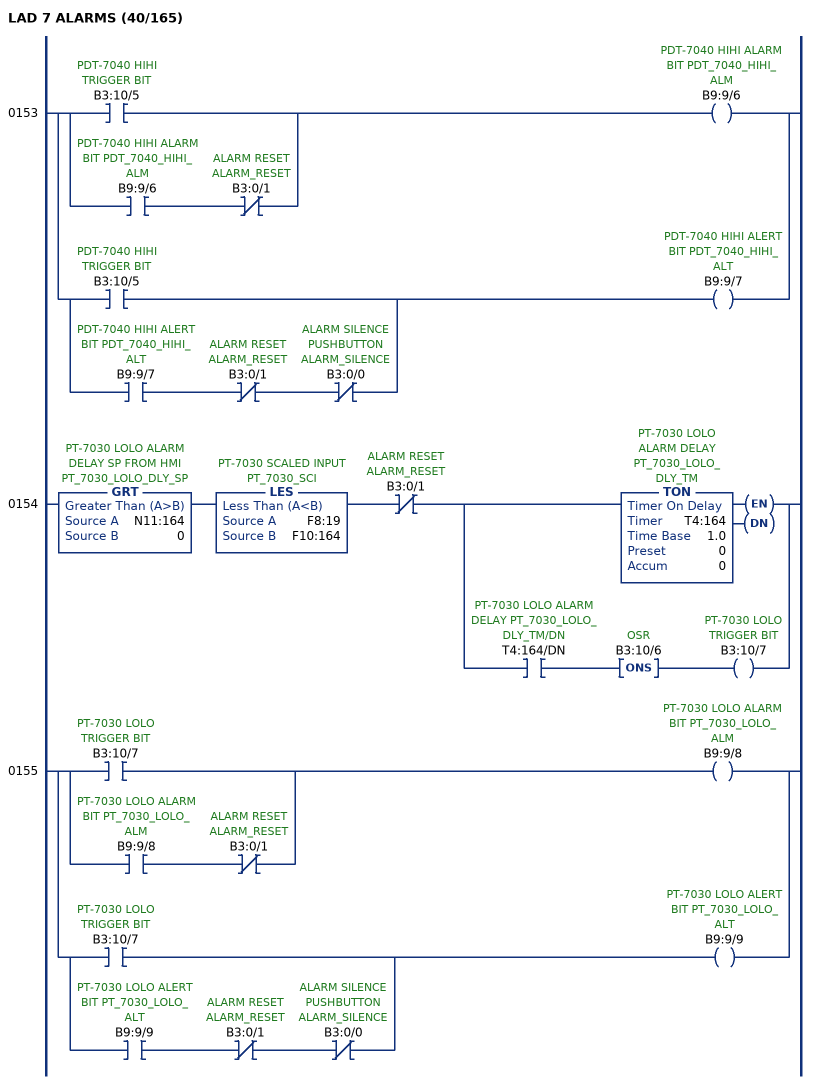
% Rung: 153 %
SOR BST BST XIC B3:10/5 NXB XIC B9:9/6 XIO B3:0/1 BND OTE B9:9/6 NXB BST XIC B3:10/5 NXB XIC B9:9/7 XIO B3:0/1 XIO B3:0/0 BND OTE B9:9/7 BND EOR
%   B3:10/5  "PDT-7040 HIHI TRIGGER BIT" %
%   B9:9/6  PDT_7040_HIHI_ALM  "PDT-7040 HIHI ALARM BIT" %
%   B3:0/1  ALARM_RESET  "ALARM RESET" %
%   B9:9/7  PDT_7040_HIHI_ALT  "PDT-7040 HIHI ALERT BIT" %
%   B3:0/0  ALARM_SILENCE  "ALARM SILENCE PUSHBUTTON" %
% Rung: 154 %
SOR GRT N11:164 0 LES F8:19 F10:164 XIO B3:0/1 BST TON T4:164 1.0 0 0 NXB XIC T4:164/DN OSR B3:10/6 OTE B3:10/7 BND EOR
%   N11:164  PT_7030_LOLO_DLY_SP  "PT-7030 LOLO ALARM DELAY SP FROM HMI" %
%   F8:19  PT_7030_SCI  "PT-7030 SCALED INPUT" %
%   F10:164  PT_7030_LOLO_SP  "PT-7030 LOLO ALARM SP" %
%   B3:0/1  ALARM_RESET  "ALARM RESET" %
%   T4:164  PT_7030_LOLO_DLY_TM  "PT-7030 LOLO ALARM DELAY" %
%   B3:10/6  "OSR" %
%   B3:10/7  "PT-7030 LOLO TRIGGER BIT" %
% Rung: 155 %
SOR BST BST XIC B3:10/7 NXB XIC B9:9/8 XIO B3:0/1 BND OTE B9:9/8 NXB BST XIC B3:10/7 NXB XIC B9:9/9 XIO B3:0/1 XIO B3:0/0 BND OTE B9:9/9 BND EOR
%   B3:10/7  "PT-7030 LOLO TRIGGER BIT" %
%   B9:9/8  PT_7030_LOLO_ALM  "PT-7030 LOLO ALARM BIT" %
%   B3:0/1  ALARM_RESET  "ALARM RESET" %
%   B9:9/9  PT_7030_LOLO_ALT  "PT-7030 LOLO ALERT BIT" %
%   B3:0/0  ALARM_SILENCE  "ALARM SILENCE PUSHBUTTON" %

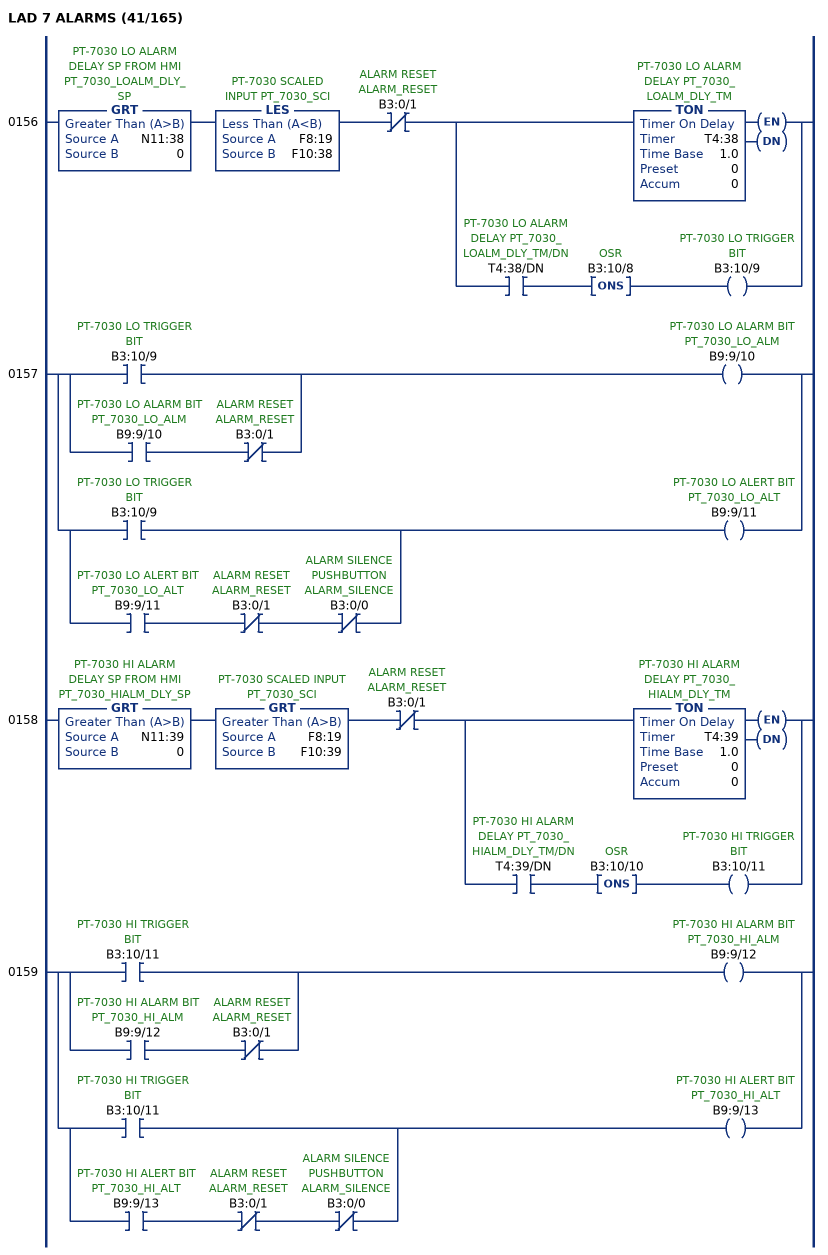
% Rung: 156 %
SOR GRT N11:38 0 LES F8:19 F10:38 XIO B3:0/1 BST TON T4:38 1.0 0 0 NXB XIC T4:38/DN OSR B3:10/8 OTE B3:10/9 BND EOR
%   N11:38  PT_7030_LOALM_DLY_SP  "PT-7030 LO ALARM DELAY SP FROM HMI" %
%   F8:19  PT_7030_SCI  "PT-7030 SCALED INPUT" %
%   F10:38  PT_7030_LOALM_SP  "PT-7030 LO ALARM SP" %
%   B3:0/1  ALARM_RESET  "ALARM RESET" %
%   T4:38  PT_7030_LOALM_DLY_TM  "PT-7030 LO ALARM DELAY" %
%   B3:10/8  "OSR" %
%   B3:10/9  "PT-7030 LO TRIGGER BIT" %
% Rung: 157 %
SOR BST BST XIC B3:10/9 NXB XIC B9:9/10 XIO B3:0/1 BND OTE B9:9/10 NXB BST XIC B3:10/9 NXB XIC B9:9/11 XIO B3:0/1 XIO B3:0/0 BND OTE B9:9/11 BND EOR
%   B3:10/9  "PT-7030 LO TRIGGER BIT" %
%   B9:9/10  PT_7030_LO_ALM  "PT-7030 LO ALARM BIT" %
%   B3:0/1  ALARM_RESET  "ALARM RESET" %
%   B9:9/11  PT_7030_LO_ALT  "PT-7030 LO ALERT BIT" %
%   B3:0/0  ALARM_SILENCE  "ALARM SILENCE PUSHBUTTON" %
% Rung: 158 %
SOR GRT N11:39 0 GRT F8:19 F10:39 XIO B3:0/1 BST TON T4:39 1.0 0 0 NXB XIC T4:39/DN OSR B3:10/10 OTE B3:10/11 BND EOR
%   N11:39  PT_7030_HIALM_DLY_SP  "PT-7030 HI ALARM DELAY SP FROM HMI" %
%   F8:19  PT_7030_SCI  "PT-7030 SCALED INPUT" %
%   F10:39  PT_7030_HIALM_SP  "PT-7030 HI ALARM SP" %
%   B3:0/1  ALARM_RESET  "ALARM RESET" %
%   T4:39  PT_7030_HIALM_DLY_TM  "PT-7030 HI ALARM DELAY" %
%   B3:10/10  "OSR" %
%   B3:10/11  "PT-7030 HI TRIGGER BIT" %
% Rung: 159 %
SOR BST BST XIC B3:10/11 NXB XIC B9:9/12 XIO B3:0/1 BND OTE B9:9/12 NXB BST XIC B3:10/11 NXB XIC B9:9/13 XIO B3:0/1 XIO B3:0/0 BND OTE B9:9/13 BND EOR
%   B3:10/11  "PT-7030 HI TRIGGER BIT" %
%   B9:9/12  PT_7030_HI_ALM  "PT-7030 HI ALARM BIT" %
%   B3:0/1  ALARM_RESET  "ALARM RESET" %
%   B9:9/13  PT_7030_HI_ALT  "PT-7030 HI ALERT BIT" %
%   B3:0/0  ALARM_SILENCE  "ALARM SILENCE PUSHBUTTON" %

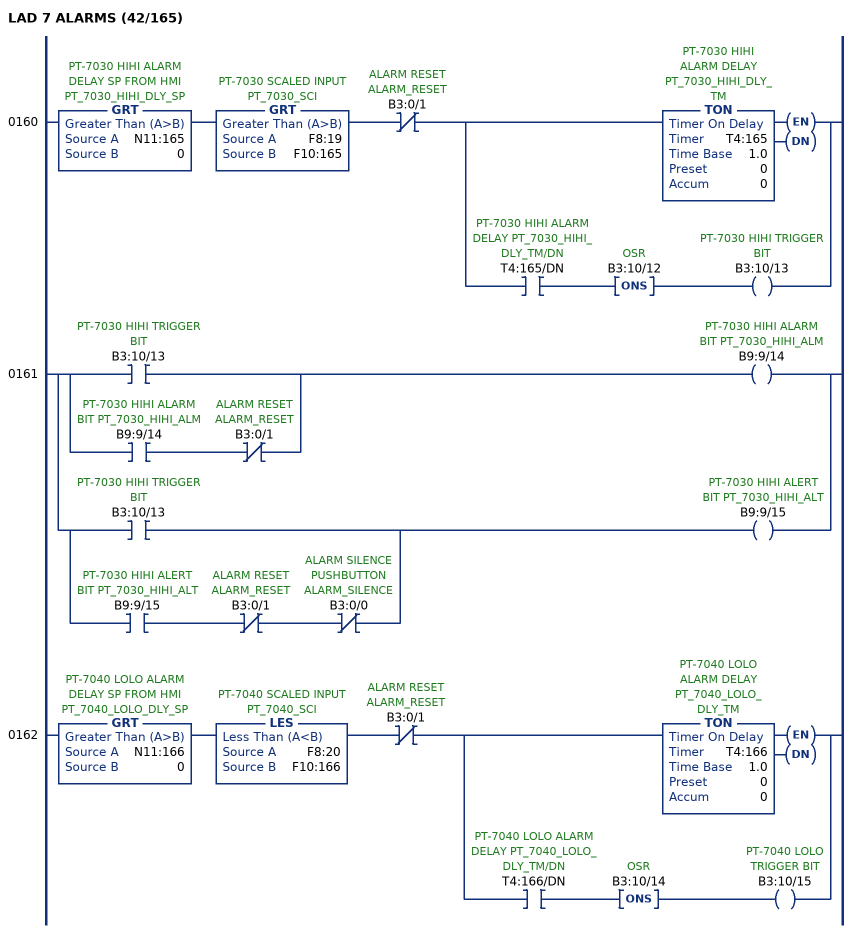
% Rung: 160 %
SOR GRT N11:165 0 GRT F8:19 F10:165 XIO B3:0/1 BST TON T4:165 1.0 0 0 NXB XIC T4:165/DN OSR B3:10/12 OTE B3:10/13 BND EOR
%   N11:165  PT_7030_HIHI_DLY_SP  "PT-7030 HIHI ALARM DELAY SP FROM HMI" %
%   F8:19  PT_7030_SCI  "PT-7030 SCALED INPUT" %
%   F10:165  PT_7030_HIHI_SP  "PT-7030 HIHI ALARM SP" %
%   B3:0/1  ALARM_RESET  "ALARM RESET" %
%   T4:165  PT_7030_HIHI_DLY_TM  "PT-7030 HIHI ALARM DELAY" %
%   B3:10/12  "OSR" %
%   B3:10/13  "PT-7030 HIHI TRIGGER BIT" %
% Rung: 161 %
SOR BST BST XIC B3:10/13 NXB XIC B9:9/14 XIO B3:0/1 BND OTE B9:9/14 NXB BST XIC B3:10/13 NXB XIC B9:9/15 XIO B3:0/1 XIO B3:0/0 BND OTE B9:9/15 BND EOR
%   B3:10/13  "PT-7030 HIHI TRIGGER BIT" %
%   B9:9/14  PT_7030_HIHI_ALM  "PT-7030 HIHI ALARM BIT" %
%   B3:0/1  ALARM_RESET  "ALARM RESET" %
%   B9:9/15  PT_7030_HIHI_ALT  "PT-7030 HIHI ALERT BIT" %
%   B3:0/0  ALARM_SILENCE  "ALARM SILENCE PUSHBUTTON" %
% Rung: 162 %
SOR GRT N11:166 0 LES F8:20 F10:166 XIO B3:0/1 BST TON T4:166 1.0 0 0 NXB XIC T4:166/DN OSR B3:10/14 OTE B3:10/15 BND EOR
%   N11:166  PT_7040_LOLO_DLY_SP  "PT-7040 LOLO ALARM DELAY SP FROM HMI" %
%   F8:20  PT_7040_SCI  "PT-7040 SCALED INPUT" %
%   F10:166  PT_7040_LOLO_SP  "PT-7040 LOLO ALARM SP" %
%   B3:0/1  ALARM_RESET  "ALARM RESET" %
%   T4:166  PT_7040_LOLO_DLY_TM  "PT-7040 LOLO ALARM DELAY" %
%   B3:10/14  "OSR" %
%   B3:10/15  "PT-7040 LOLO TRIGGER BIT" %

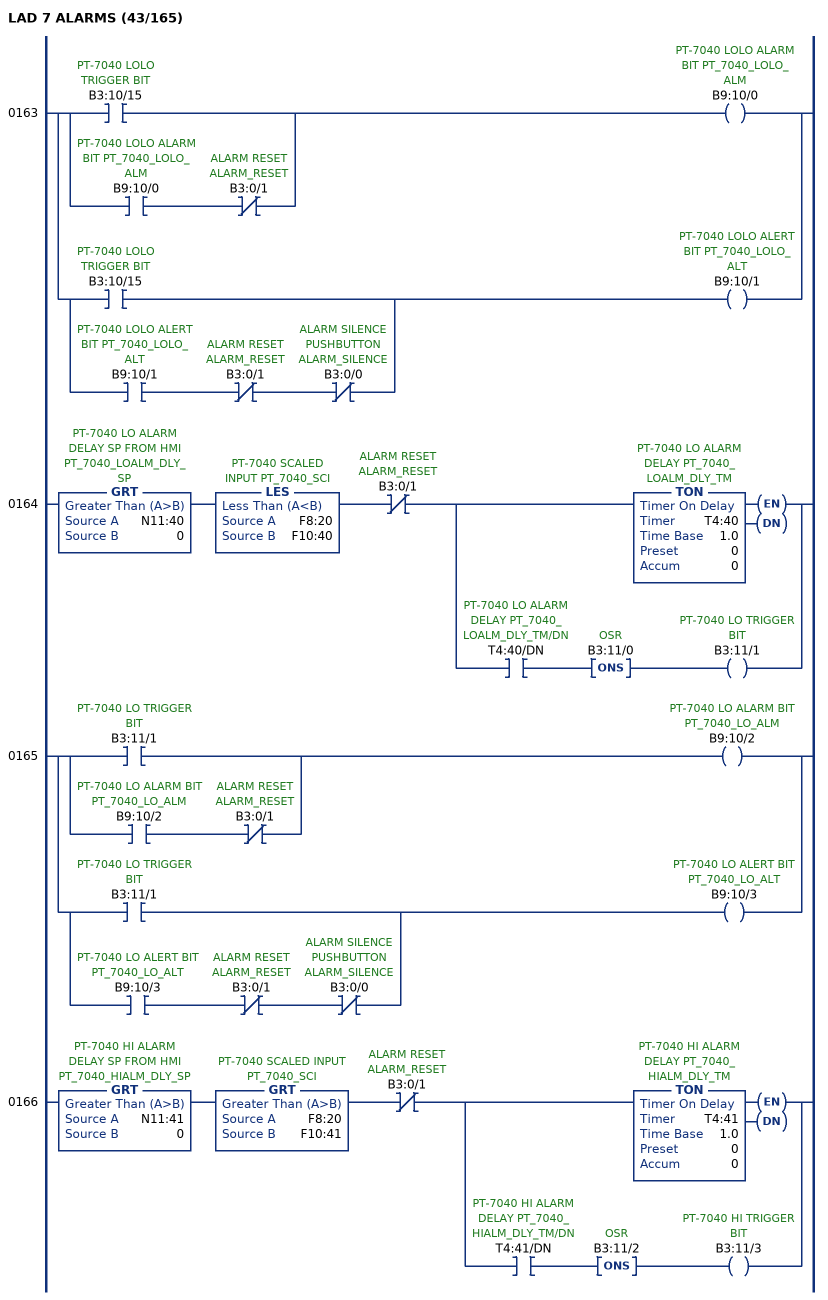
% Rung: 163 %
SOR BST BST XIC B3:10/15 NXB XIC B9:10/0 XIO B3:0/1 BND OTE B9:10/0 NXB BST XIC B3:10/15 NXB XIC B9:10/1 XIO B3:0/1 XIO B3:0/0 BND OTE B9:10/1 BND EOR
%   B3:10/15  "PT-7040 LOLO TRIGGER BIT" %
%   B9:10/0  PT_7040_LOLO_ALM  "PT-7040 LOLO ALARM BIT" %
%   B3:0/1  ALARM_RESET  "ALARM RESET" %
%   B9:10/1  PT_7040_LOLO_ALT  "PT-7040 LOLO ALERT BIT" %
%   B3:0/0  ALARM_SILENCE  "ALARM SILENCE PUSHBUTTON" %
% Rung: 164 %
SOR GRT N11:40 0 LES F8:20 F10:40 XIO B3:0/1 BST TON T4:40 1.0 0 0 NXB XIC T4:40/DN OSR B3:11/0 OTE B3:11/1 BND EOR
%   N11:40  PT_7040_LOALM_DLY_SP  "PT-7040 LO ALARM DELAY SP FROM HMI" %
%   F8:20  PT_7040_SCI  "PT-7040 SCALED INPUT" %
%   F10:40  PT_7040_LOALM_SP  "PT-7040 LO ALARM SP" %
%   B3:0/1  ALARM_RESET  "ALARM RESET" %
%   T4:40  PT_7040_LOALM_DLY_TM  "PT-7040 LO ALARM DELAY" %
%   B3:11/0  "OSR" %
%   B3:11/1  "PT-7040 LO TRIGGER BIT" %
% Rung: 165 %
SOR BST BST XIC B3:11/1 NXB XIC B9:10/2 XIO B3:0/1 BND OTE B9:10/2 NXB BST XIC B3:11/1 NXB XIC B9:10/3 XIO B3:0/1 XIO B3:0/0 BND OTE B9:10/3 BND EOR
%   B3:11/1  "PT-7040 LO TRIGGER BIT" %
%   B9:10/2  PT_7040_LO_ALM  "PT-7040 LO ALARM BIT" %
%   B3:0/1  ALARM_RESET  "ALARM RESET" %
%   B9:10/3  PT_7040_LO_ALT  "PT-7040 LO ALERT BIT" %
%   B3:0/0  ALARM_SILENCE  "ALARM SILENCE PUSHBUTTON" %
% Rung: 166 %
SOR GRT N11:41 0 GRT F8:20 F10:41 XIO B3:0/1 BST TON T4:41 1.0 0 0 NXB XIC T4:41/DN OSR B3:11/2 OTE B3:11/3 BND EOR
%   N11:41  PT_7040_HIALM_DLY_SP  "PT-7040 HI ALARM DELAY SP FROM HMI" %
%   F8:20  PT_7040_SCI  "PT-7040 SCALED INPUT" %
%   F10:41  PT_7040_HIALM_SP  "PT-7040 HI ALARM SP" %
%   B3:0/1  ALARM_RESET  "ALARM RESET" %
%   T4:41  PT_7040_HIALM_DLY_TM  "PT-7040 HI ALARM DELAY" %
%   B3:11/2  "OSR" %
%   B3:11/3  "PT-7040 HI TRIGGER BIT" %

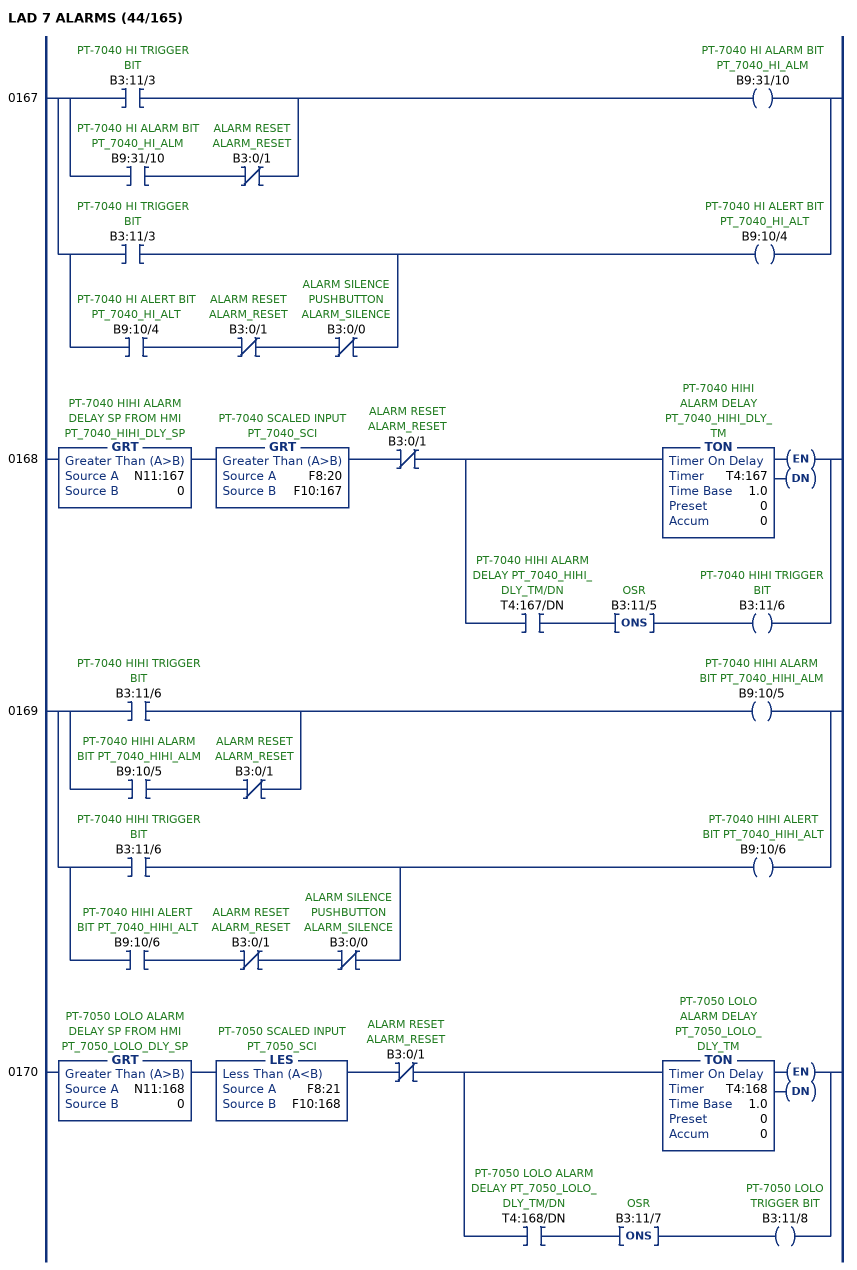
% Rung: 167 %
SOR BST BST XIC B3:11/3 NXB XIC B9:31/10 XIO B3:0/1 BND OTE B9:31/10 NXB BST XIC B3:11/3 NXB XIC B9:10/4 XIO B3:0/1 XIO B3:0/0 BND OTE B9:10/4 BND EOR
%   B3:11/3  "PT-7040 HI TRIGGER BIT" %
%   B9:31/10  PT_7040_HI_ALM  "PT-7040 HI ALARM BIT" %
%   B3:0/1  ALARM_RESET  "ALARM RESET" %
%   B9:10/4  PT_7040_HI_ALT  "PT-7040 HI ALERT BIT" %
%   B3:0/0  ALARM_SILENCE  "ALARM SILENCE PUSHBUTTON" %
% Rung: 168 %
SOR GRT N11:167 0 GRT F8:20 F10:167 XIO B3:0/1 BST TON T4:167 1.0 0 0 NXB XIC T4:167/DN OSR B3:11/5 OTE B3:11/6 BND EOR
%   N11:167  PT_7040_HIHI_DLY_SP  "PT-7040 HIHI ALARM DELAY SP FROM HMI" %
%   F8:20  PT_7040_SCI  "PT-7040 SCALED INPUT" %
%   F10:167  PT_7040_HIHI_SP  "PT-7040 HIHI ALARM SP" %
%   B3:0/1  ALARM_RESET  "ALARM RESET" %
%   T4:167  PT_7040_HIHI_DLY_TM  "PT-7040 HIHI ALARM DELAY" %
%   B3:11/5  "OSR" %
%   B3:11/6  "PT-7040 HIHI TRIGGER BIT" %
% Rung: 169 %
SOR BST BST XIC B3:11/6 NXB XIC B9:10/5 XIO B3:0/1 BND OTE B9:10/5 NXB BST XIC B3:11/6 NXB XIC B9:10/6 XIO B3:0/1 XIO B3:0/0 BND OTE B9:10/6 BND EOR
%   B3:11/6  "PT-7040 HIHI TRIGGER BIT" %
%   B9:10/5  PT_7040_HIHI_ALM  "PT-7040 HIHI ALARM BIT" %
%   B3:0/1  ALARM_RESET  "ALARM RESET" %
%   B9:10/6  PT_7040_HIHI_ALT  "PT-7040 HIHI ALERT BIT" %
%   B3:0/0  ALARM_SILENCE  "ALARM SILENCE PUSHBUTTON" %
% Rung: 170 %
SOR GRT N11:168 0 LES F8:21 F10:168 XIO B3:0/1 BST TON T4:168 1.0 0 0 NXB XIC T4:168/DN OSR B3:11/7 OTE B3:11/8 BND EOR
%   N11:168  PT_7050_LOLO_DLY_SP  "PT-7050 LOLO ALARM DELAY SP FROM HMI" %
%   F8:21  PT_7050_SCI  "PT-7050 SCALED INPUT" %
%   F10:168  PT_7050_LOLO_SP  "PT-7050 LOLO ALARM SP" %
%   B3:0/1  ALARM_RESET  "ALARM RESET" %
%   T4:168  PT_7050_LOLO_DLY_TM  "PT-7050 LOLO ALARM DELAY" %
%   B3:11/7  "OSR" %
%   B3:11/8  "PT-7050 LOLO TRIGGER BIT" %

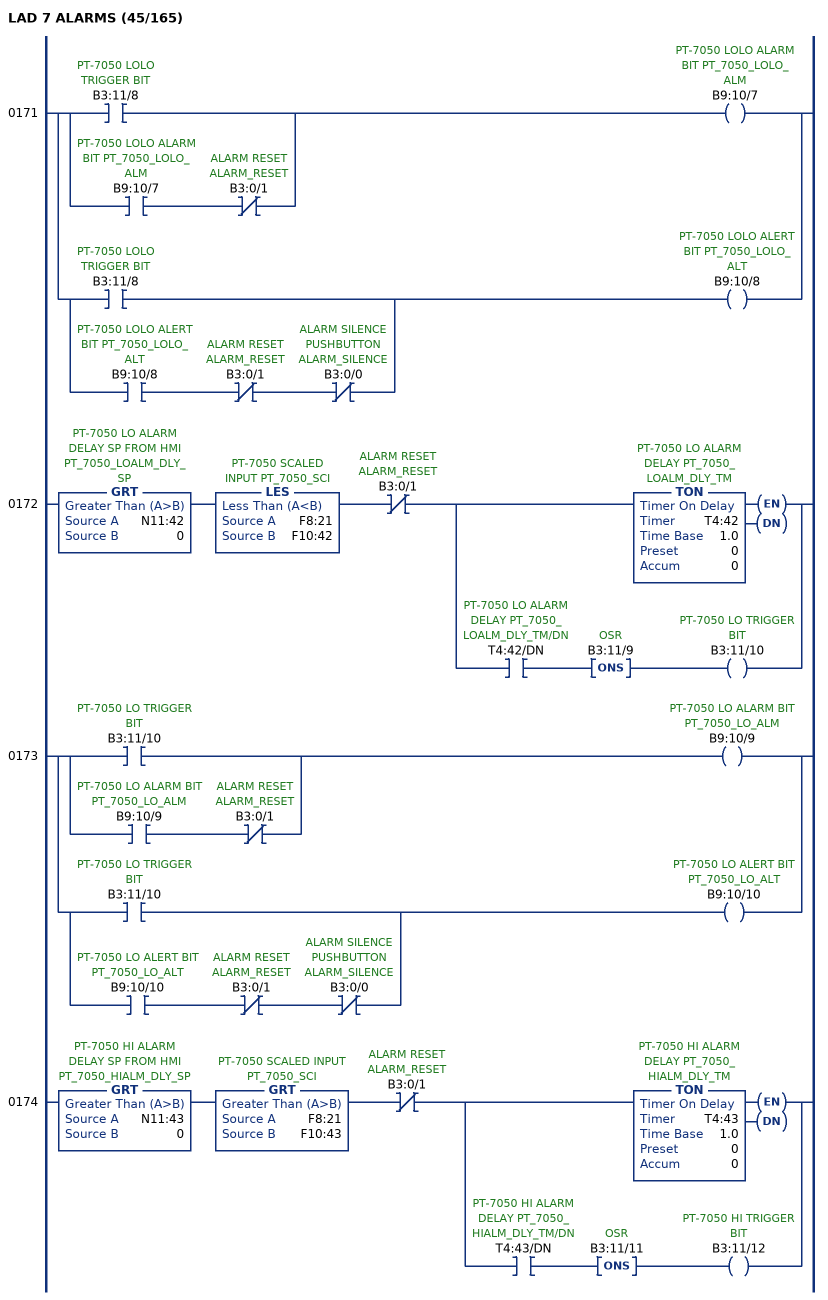
% Rung: 171 %
SOR BST BST XIC B3:11/8 NXB XIC B9:10/7 XIO B3:0/1 BND OTE B9:10/7 NXB BST XIC B3:11/8 NXB XIC B9:10/8 XIO B3:0/1 XIO B3:0/0 BND OTE B9:10/8 BND EOR
%   B3:11/8  "PT-7050 LOLO TRIGGER BIT" %
%   B9:10/7  PT_7050_LOLO_ALM  "PT-7050 LOLO ALARM BIT" %
%   B3:0/1  ALARM_RESET  "ALARM RESET" %
%   B9:10/8  PT_7050_LOLO_ALT  "PT-7050 LOLO ALERT BIT" %
%   B3:0/0  ALARM_SILENCE  "ALARM SILENCE PUSHBUTTON" %
% Rung: 172 %
SOR GRT N11:42 0 LES F8:21 F10:42 XIO B3:0/1 BST TON T4:42 1.0 0 0 NXB XIC T4:42/DN OSR B3:11/9 OTE B3:11/10 BND EOR
%   N11:42  PT_7050_LOALM_DLY_SP  "PT-7050 LO ALARM DELAY SP FROM HMI" %
%   F8:21  PT_7050_SCI  "PT-7050 SCALED INPUT" %
%   F10:42  PT_7050_LOALM_SP  "PT-7050 LO ALARM SP" %
%   B3:0/1  ALARM_RESET  "ALARM RESET" %
%   T4:42  PT_7050_LOALM_DLY_TM  "PT-7050 LO ALARM DELAY" %
%   B3:11/9  "OSR" %
%   B3:11/10  "PT-7050 LO TRIGGER BIT" %
% Rung: 173 %
SOR BST BST XIC B3:11/10 NXB XIC B9:10/9 XIO B3:0/1 BND OTE B9:10/9 NXB BST XIC B3:11/10 NXB XIC B9:10/10 XIO B3:0/1 XIO B3:0/0 BND OTE B9:10/10 BND EOR
%   B3:11/10  "PT-7050 LO TRIGGER BIT" %
%   B9:10/9  PT_7050_LO_ALM  "PT-7050 LO ALARM BIT" %
%   B3:0/1  ALARM_RESET  "ALARM RESET" %
%   B9:10/10  PT_7050_LO_ALT  "PT-7050 LO ALERT BIT" %
%   B3:0/0  ALARM_SILENCE  "ALARM SILENCE PUSHBUTTON" %
% Rung: 174 %
SOR GRT N11:43 0 GRT F8:21 F10:43 XIO B3:0/1 BST TON T4:43 1.0 0 0 NXB XIC T4:43/DN OSR B3:11/11 OTE B3:11/12 BND EOR
%   N11:43  PT_7050_HIALM_DLY_SP  "PT-7050 HI ALARM DELAY SP FROM HMI" %
%   F8:21  PT_7050_SCI  "PT-7050 SCALED INPUT" %
%   F10:43  PT_7050_HIALM_SP  "PT-7050 HI ALARM SP" %
%   B3:0/1  ALARM_RESET  "ALARM RESET" %
%   T4:43  PT_7050_HIALM_DLY_TM  "PT-7050 HI ALARM DELAY" %
%   B3:11/11  "OSR" %
%   B3:11/12  "PT-7050 HI TRIGGER BIT" %

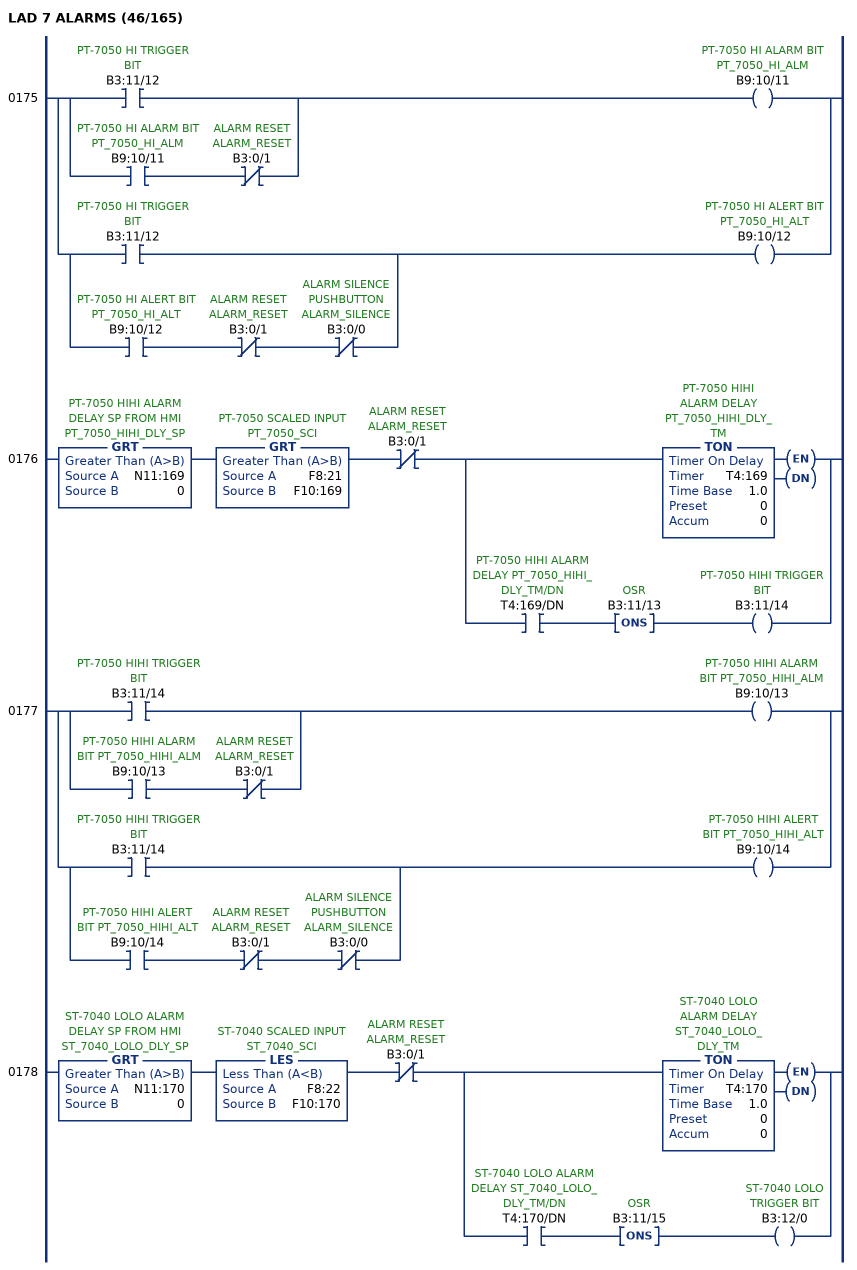
% Rung: 175 %
SOR BST BST XIC B3:11/12 NXB XIC B9:10/11 XIO B3:0/1 BND OTE B9:10/11 NXB BST XIC B3:11/12 NXB XIC B9:10/12 XIO B3:0/1 XIO B3:0/0 BND OTE B9:10/12 BND EOR
%   B3:11/12  "PT-7050 HI TRIGGER BIT" %
%   B9:10/11  PT_7050_HI_ALM  "PT-7050 HI ALARM BIT" %
%   B3:0/1  ALARM_RESET  "ALARM RESET" %
%   B9:10/12  PT_7050_HI_ALT  "PT-7050 HI ALERT BIT" %
%   B3:0/0  ALARM_SILENCE  "ALARM SILENCE PUSHBUTTON" %
% Rung: 176 %
SOR GRT N11:169 0 GRT F8:21 F10:169 XIO B3:0/1 BST TON T4:169 1.0 0 0 NXB XIC T4:169/DN OSR B3:11/13 OTE B3:11/14 BND EOR
%   N11:169  PT_7050_HIHI_DLY_SP  "PT-7050 HIHI ALARM DELAY SP FROM HMI" %
%   F8:21  PT_7050_SCI  "PT-7050 SCALED INPUT" %
%   F10:169  PT_7050_HIHI_SP  "PT-7050 HIHI ALARM SP" %
%   B3:0/1  ALARM_RESET  "ALARM RESET" %
%   T4:169  PT_7050_HIHI_DLY_TM  "PT-7050 HIHI ALARM DELAY" %
%   B3:11/13  "OSR" %
%   B3:11/14  "PT-7050 HIHI TRIGGER BIT" %
% Rung: 177 %
SOR BST BST XIC B3:11/14 NXB XIC B9:10/13 XIO B3:0/1 BND OTE B9:10/13 NXB BST XIC B3:11/14 NXB XIC B9:10/14 XIO B3:0/1 XIO B3:0/0 BND OTE B9:10/14 BND EOR
%   B3:11/14  "PT-7050 HIHI TRIGGER BIT" %
%   B9:10/13  PT_7050_HIHI_ALM  "PT-7050 HIHI ALARM BIT" %
%   B3:0/1  ALARM_RESET  "ALARM RESET" %
%   B9:10/14  PT_7050_HIHI_ALT  "PT-7050 HIHI ALERT BIT" %
%   B3:0/0  ALARM_SILENCE  "ALARM SILENCE PUSHBUTTON" %
% Rung: 178 %
SOR GRT N11:170 0 LES F8:22 F10:170 XIO B3:0/1 BST TON T4:170 1.0 0 0 NXB XIC T4:170/DN OSR B3:11/15 OTE B3:12/0 BND EOR
%   N11:170  ST_7040_LOLO_DLY_SP  "ST-7040 LOLO ALARM DELAY SP FROM HMI" %
%   F8:22  ST_7040_SCI  "ST-7040 SCALED INPUT" %
%   F10:170  ST_7040_LOLO_SP  "ST-7040 LOLO ALARM SP" %
%   B3:0/1  ALARM_RESET  "ALARM RESET" %
%   T4:170  ST_7040_LOLO_DLY_TM  "ST-7040 LOLO ALARM DELAY" %
%   B3:11/15  "OSR" %
%   B3:12/0  "ST-7040 LOLO TRIGGER BIT" %

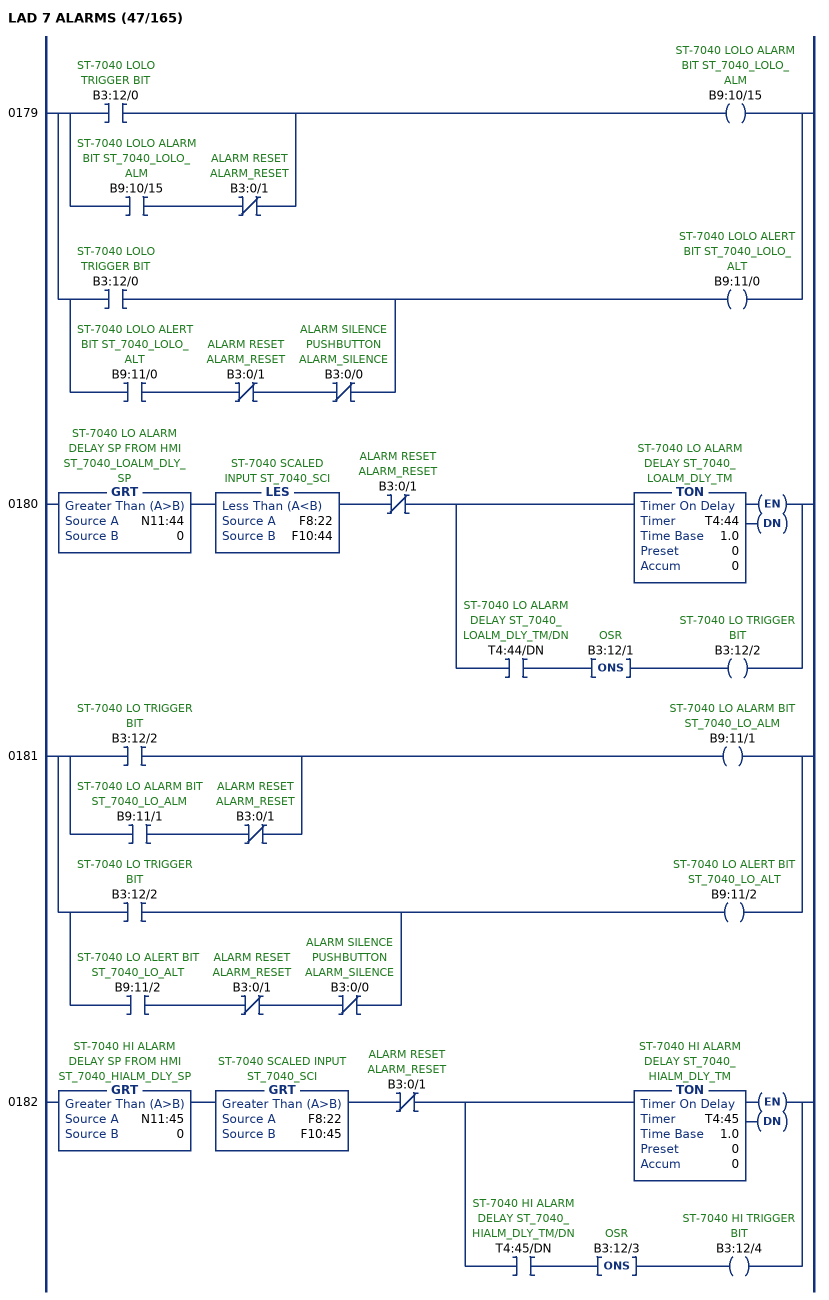
% Rung: 179 %
SOR BST BST XIC B3:12/0 NXB XIC B9:10/15 XIO B3:0/1 BND OTE B9:10/15 NXB BST XIC B3:12/0 NXB XIC B9:11/0 XIO B3:0/1 XIO B3:0/0 BND OTE B9:11/0 BND EOR
%   B3:12/0  "ST-7040 LOLO TRIGGER BIT" %
%   B9:10/15  ST_7040_LOLO_ALM  "ST-7040 LOLO ALARM BIT" %
%   B3:0/1  ALARM_RESET  "ALARM RESET" %
%   B9:11/0  ST_7040_LOLO_ALT  "ST-7040 LOLO ALERT BIT" %
%   B3:0/0  ALARM_SILENCE  "ALARM SILENCE PUSHBUTTON" %
% Rung: 180 %
SOR GRT N11:44 0 LES F8:22 F10:44 XIO B3:0/1 BST TON T4:44 1.0 0 0 NXB XIC T4:44/DN OSR B3:12/1 OTE B3:12/2 BND EOR
%   N11:44  ST_7040_LOALM_DLY_SP  "ST-7040 LO ALARM DELAY SP FROM HMI" %
%   F8:22  ST_7040_SCI  "ST-7040 SCALED INPUT" %
%   F10:44  ST_7040_LOALM_SP  "ST-7040 LO ALARM SP" %
%   B3:0/1  ALARM_RESET  "ALARM RESET" %
%   T4:44  ST_7040_LOALM_DLY_TM  "ST-7040 LO ALARM DELAY" %
%   B3:12/1  "OSR" %
%   B3:12/2  "ST-7040 LO TRIGGER BIT" %
% Rung: 181 %
SOR BST BST XIC B3:12/2 NXB XIC B9:11/1 XIO B3:0/1 BND OTE B9:11/1 NXB BST XIC B3:12/2 NXB XIC B9:11/2 XIO B3:0/1 XIO B3:0/0 BND OTE B9:11/2 BND EOR
%   B3:12/2  "ST-7040 LO TRIGGER BIT" %
%   B9:11/1  ST_7040_LO_ALM  "ST-7040 LO ALARM BIT" %
%   B3:0/1  ALARM_RESET  "ALARM RESET" %
%   B9:11/2  ST_7040_LO_ALT  "ST-7040 LO ALERT BIT" %
%   B3:0/0  ALARM_SILENCE  "ALARM SILENCE PUSHBUTTON" %
% Rung: 182 %
SOR GRT N11:45 0 GRT F8:22 F10:45 XIO B3:0/1 BST TON T4:45 1.0 0 0 NXB XIC T4:45/DN OSR B3:12/3 OTE B3:12/4 BND EOR
%   N11:45  ST_7040_HIALM_DLY_SP  "ST-7040 HI ALARM DELAY SP FROM HMI" %
%   F8:22  ST_7040_SCI  "ST-7040 SCALED INPUT" %
%   F10:45  ST_7040_HIALM_SP  "ST-7040 HI ALARM SP" %
%   B3:0/1  ALARM_RESET  "ALARM RESET" %
%   T4:45  ST_7040_HIALM_DLY_TM  "ST-7040 HI ALARM DELAY" %
%   B3:12/3  "OSR" %
%   B3:12/4  "ST-7040 HI TRIGGER BIT" %

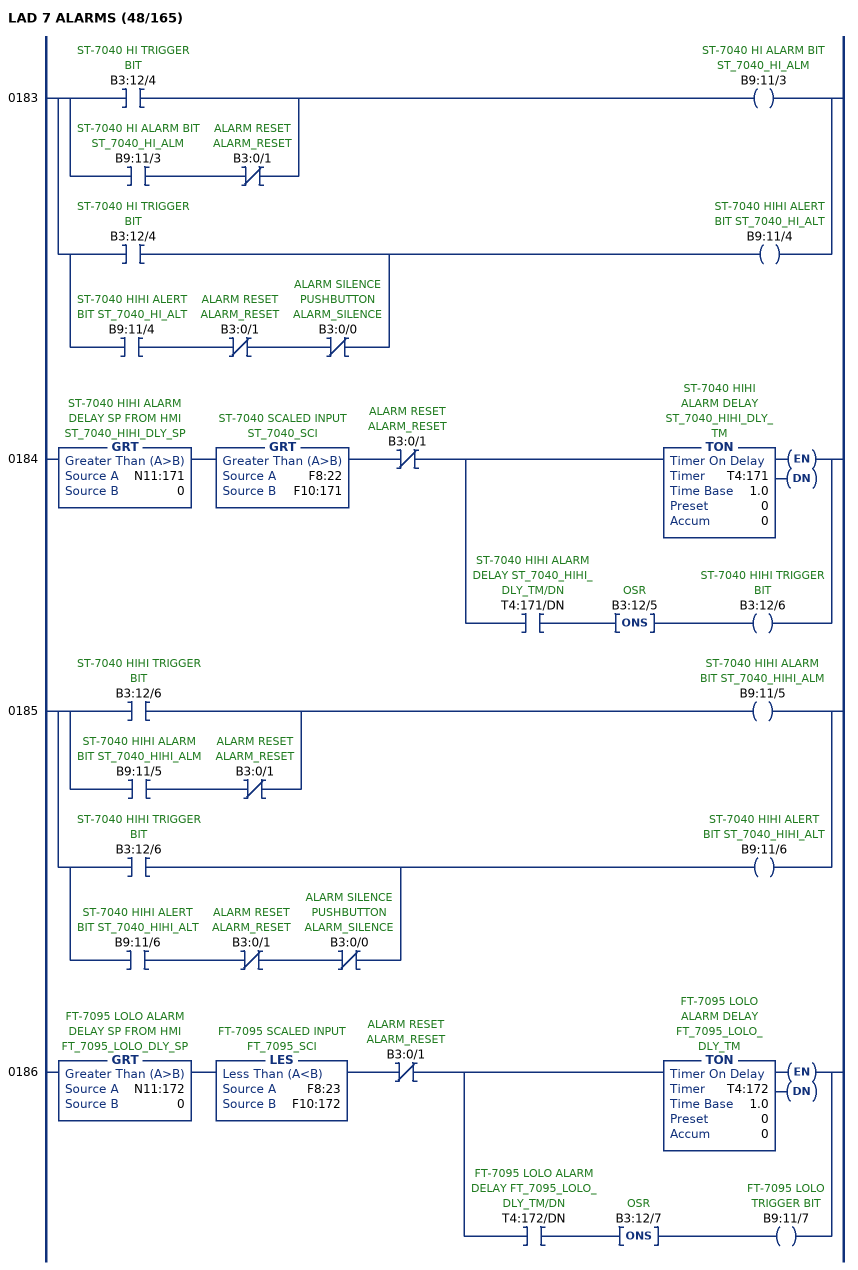
% Rung: 183 %
SOR BST BST XIC B3:12/4 NXB XIC B9:11/3 XIO B3:0/1 BND OTE B9:11/3 NXB BST XIC B3:12/4 NXB XIC B9:11/4 XIO B3:0/1 XIO B3:0/0 BND OTE B9:11/4 BND EOR
%   B3:12/4  "ST-7040 HI TRIGGER BIT" %
%   B9:11/3  ST_7040_HI_ALM  "ST-7040 HI ALARM BIT" %
%   B3:0/1  ALARM_RESET  "ALARM RESET" %
%   B9:11/4  ST_7040_HI_ALT  "ST-7040 HIHI ALERT BIT" %
%   B3:0/0  ALARM_SILENCE  "ALARM SILENCE PUSHBUTTON" %
% Rung: 184 %
SOR GRT N11:171 0 GRT F8:22 F10:171 XIO B3:0/1 BST TON T4:171 1.0 0 0 NXB XIC T4:171/DN OSR B3:12/5 OTE B3:12/6 BND EOR
%   N11:171  ST_7040_HIHI_DLY_SP  "ST-7040 HIHI ALARM DELAY SP FROM HMI" %
%   F8:22  ST_7040_SCI  "ST-7040 SCALED INPUT" %
%   F10:171  ST_7040_HIHI_SP  "ST-7040 HIHI ALARM SP" %
%   B3:0/1  ALARM_RESET  "ALARM RESET" %
%   T4:171  ST_7040_HIHI_DLY_TM  "ST-7040 HIHI ALARM DELAY" %
%   B3:12/5  "OSR" %
%   B3:12/6  "ST-7040 HIHI TRIGGER BIT" %
% Rung: 185 %
SOR BST BST XIC B3:12/6 NXB XIC B9:11/5 XIO B3:0/1 BND OTE B9:11/5 NXB BST XIC B3:12/6 NXB XIC B9:11/6 XIO B3:0/1 XIO B3:0/0 BND OTE B9:11/6 BND EOR
%   B3:12/6  "ST-7040 HIHI TRIGGER BIT" %
%   B9:11/5  ST_7040_HIHI_ALM  "ST-7040 HIHI ALARM BIT" %
%   B3:0/1  ALARM_RESET  "ALARM RESET" %
%   B9:11/6  ST_7040_HIHI_ALT  "ST-7040 HIHI ALERT BIT" %
%   B3:0/0  ALARM_SILENCE  "ALARM SILENCE PUSHBUTTON" %
% Rung: 186 %
SOR GRT N11:172 0 LES F8:23 F10:172 XIO B3:0/1 BST TON T4:172 1.0 0 0 NXB XIC T4:172/DN OSR B3:12/7 OTE B9:11/7 BND EOR
%   N11:172  FT_7095_LOLO_DLY_SP  "FT-7095 LOLO ALARM DELAY SP FROM HMI" %
%   F8:23  FT_7095_SCI  "FT-7095 SCALED INPUT" %
%   F10:172  FT_7095_LOLO_SP  "FT-7095 LOLO ALARM SP" %
%   B3:0/1  ALARM_RESET  "ALARM RESET" %
%   T4:172  FT_7095_LOLO_DLY_TM  "FT-7095 LOLO ALARM DELAY" %
%   B3:12/7  "OSR" %
%   B9:11/7  "FT-7095 LOLO TRIGGER BIT" %

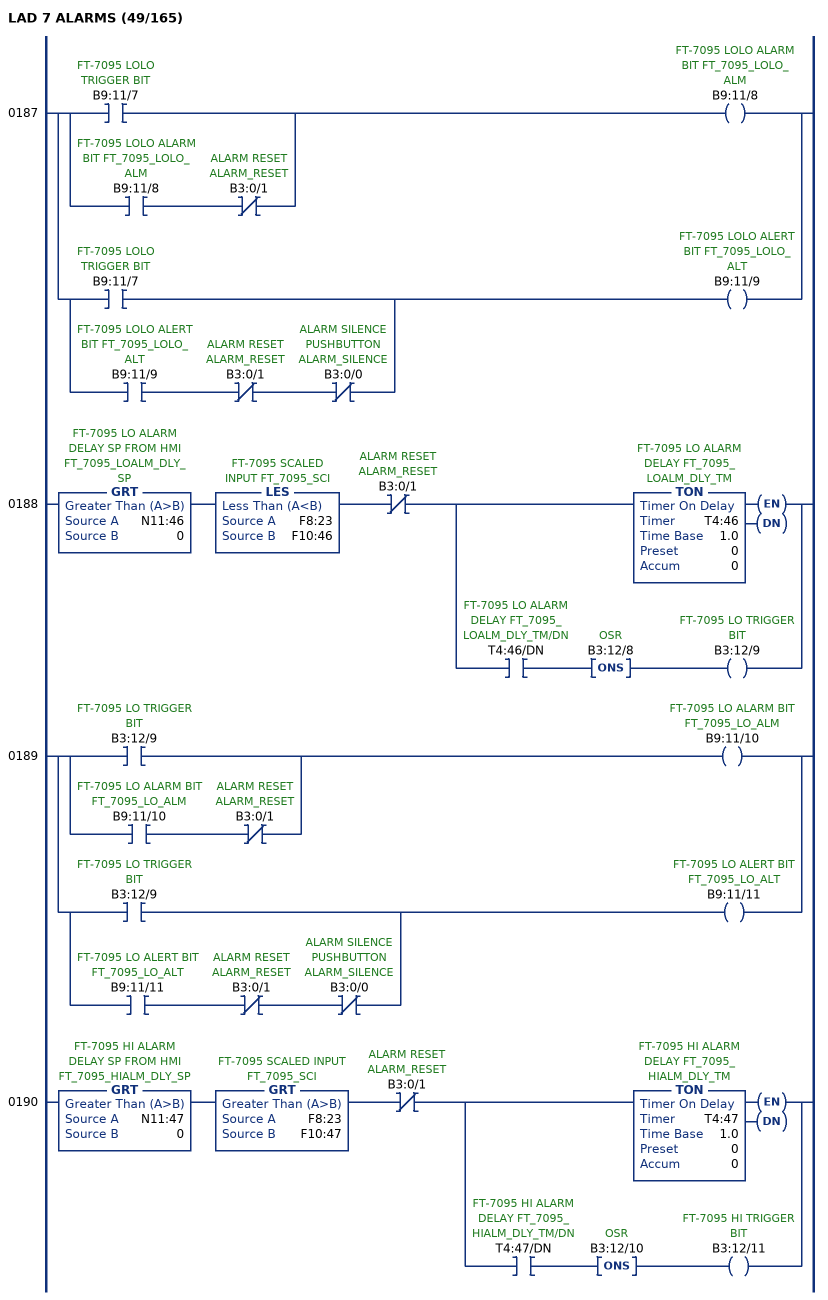
% Rung: 187 %
SOR BST BST XIC B9:11/7 NXB XIC B9:11/8 XIO B3:0/1 BND OTE B9:11/8 NXB BST XIC B9:11/7 NXB XIC B9:11/9 XIO B3:0/1 XIO B3:0/0 BND OTE B9:11/9 BND EOR
%   B9:11/7  "FT-7095 LOLO TRIGGER BIT" %
%   B9:11/8  FT_7095_LOLO_ALM  "FT-7095 LOLO ALARM BIT" %
%   B3:0/1  ALARM_RESET  "ALARM RESET" %
%   B9:11/9  FT_7095_LOLO_ALT  "FT-7095 LOLO ALERT BIT" %
%   B3:0/0  ALARM_SILENCE  "ALARM SILENCE PUSHBUTTON" %
% Rung: 188 %
SOR GRT N11:46 0 LES F8:23 F10:46 XIO B3:0/1 BST TON T4:46 1.0 0 0 NXB XIC T4:46/DN OSR B3:12/8 OTE B3:12/9 BND EOR
%   N11:46  FT_7095_LOALM_DLY_SP  "FT-7095 LO ALARM DELAY SP FROM HMI" %
%   F8:23  FT_7095_SCI  "FT-7095 SCALED INPUT" %
%   F10:46  FT_7095_LOALM_SP  "FT-7095 LO ALARM SP" %
%   B3:0/1  ALARM_RESET  "ALARM RESET" %
%   T4:46  FT_7095_LOALM_DLY_TM  "FT-7095 LO ALARM DELAY" %
%   B3:12/8  "OSR" %
%   B3:12/9  "FT-7095 LO TRIGGER BIT" %
% Rung: 189 %
SOR BST BST XIC B3:12/9 NXB XIC B9:11/10 XIO B3:0/1 BND OTE B9:11/10 NXB BST XIC B3:12/9 NXB XIC B9:11/11 XIO B3:0/1 XIO B3:0/0 BND OTE B9:11/11 BND EOR
%   B3:12/9  "FT-7095 LO TRIGGER BIT" %
%   B9:11/10  FT_7095_LO_ALM  "FT-7095 LO ALARM BIT" %
%   B3:0/1  ALARM_RESET  "ALARM RESET" %
%   B9:11/11  FT_7095_LO_ALT  "FT-7095 LO ALERT BIT" %
%   B3:0/0  ALARM_SILENCE  "ALARM SILENCE PUSHBUTTON" %
% Rung: 190 %
SOR GRT N11:47 0 GRT F8:23 F10:47 XIO B3:0/1 BST TON T4:47 1.0 0 0 NXB XIC T4:47/DN OSR B3:12/10 OTE B3:12/11 BND EOR
%   N11:47  FT_7095_HIALM_DLY_SP  "FT-7095 HI ALARM DELAY SP FROM HMI" %
%   F8:23  FT_7095_SCI  "FT-7095 SCALED INPUT" %
%   F10:47  FT_7095_HIALM_SP  "FT-7095 HI ALARM SP" %
%   B3:0/1  ALARM_RESET  "ALARM RESET" %
%   T4:47  FT_7095_HIALM_DLY_TM  "FT-7095 HI ALARM DELAY" %
%   B3:12/10  "OSR" %
%   B3:12/11  "FT-7095 HI TRIGGER BIT" %

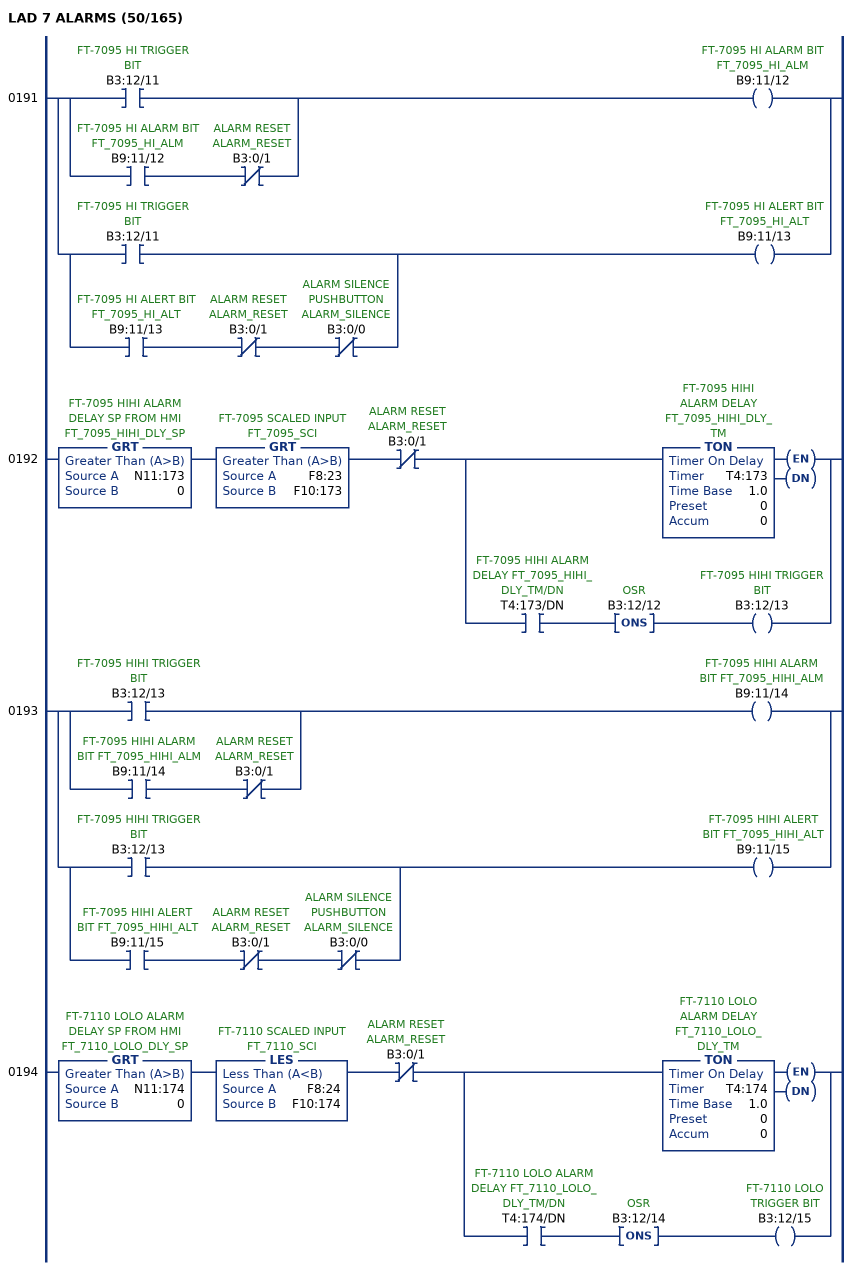
% Rung: 191 %
SOR BST BST XIC B3:12/11 NXB XIC B9:11/12 XIO B3:0/1 BND OTE B9:11/12 NXB BST XIC B3:12/11 NXB XIC B9:11/13 XIO B3:0/1 XIO B3:0/0 BND OTE B9:11/13 BND EOR
%   B3:12/11  "FT-7095 HI TRIGGER BIT" %
%   B9:11/12  FT_7095_HI_ALM  "FT-7095 HI ALARM BIT" %
%   B3:0/1  ALARM_RESET  "ALARM RESET" %
%   B9:11/13  FT_7095_HI_ALT  "FT-7095 HI ALERT BIT" %
%   B3:0/0  ALARM_SILENCE  "ALARM SILENCE PUSHBUTTON" %
% Rung: 192 %
SOR GRT N11:173 0 GRT F8:23 F10:173 XIO B3:0/1 BST TON T4:173 1.0 0 0 NXB XIC T4:173/DN OSR B3:12/12 OTE B3:12/13 BND EOR
%   N11:173  FT_7095_HIHI_DLY_SP  "FT-7095 HIHI ALARM DELAY SP FROM HMI" %
%   F8:23  FT_7095_SCI  "FT-7095 SCALED INPUT" %
%   F10:173  FT_7095_HIHI_SP  "FT-7095 HIHI ALARM SP" %
%   B3:0/1  ALARM_RESET  "ALARM RESET" %
%   T4:173  FT_7095_HIHI_DLY_TM  "FT-7095 HIHI ALARM DELAY" %
%   B3:12/12  "OSR" %
%   B3:12/13  "FT-7095 HIHI TRIGGER BIT" %
% Rung: 193 %
SOR BST BST XIC B3:12/13 NXB XIC B9:11/14 XIO B3:0/1 BND OTE B9:11/14 NXB BST XIC B3:12/13 NXB XIC B9:11/15 XIO B3:0/1 XIO B3:0/0 BND OTE B9:11/15 BND EOR
%   B3:12/13  "FT-7095 HIHI TRIGGER BIT" %
%   B9:11/14  FT_7095_HIHI_ALM  "FT-7095 HIHI ALARM BIT" %
%   B3:0/1  ALARM_RESET  "ALARM RESET" %
%   B9:11/15  FT_7095_HIHI_ALT  "FT-7095 HIHI ALERT BIT" %
%   B3:0/0  ALARM_SILENCE  "ALARM SILENCE PUSHBUTTON" %
% Rung: 194 %
SOR GRT N11:174 0 LES F8:24 F10:174 XIO B3:0/1 BST TON T4:174 1.0 0 0 NXB XIC T4:174/DN OSR B3:12/14 OTE B3:12/15 BND EOR
%   N11:174  FT_7110_LOLO_DLY_SP  "FT-7110 LOLO ALARM DELAY SP FROM HMI" %
%   F8:24  FT_7110_SCI  "FT-7110 SCALED INPUT" %
%   F10:174  FT_7110_LOLO_SP  "FT-7110 LOLO ALARM SP" %
%   B3:0/1  ALARM_RESET  "ALARM RESET" %
%   T4:174  FT_7110_LOLO_DLY_TM  "FT-7110 LOLO ALARM DELAY" %
%   B3:12/14  "OSR" %
%   B3:12/15  "FT-7110 LOLO TRIGGER BIT" %

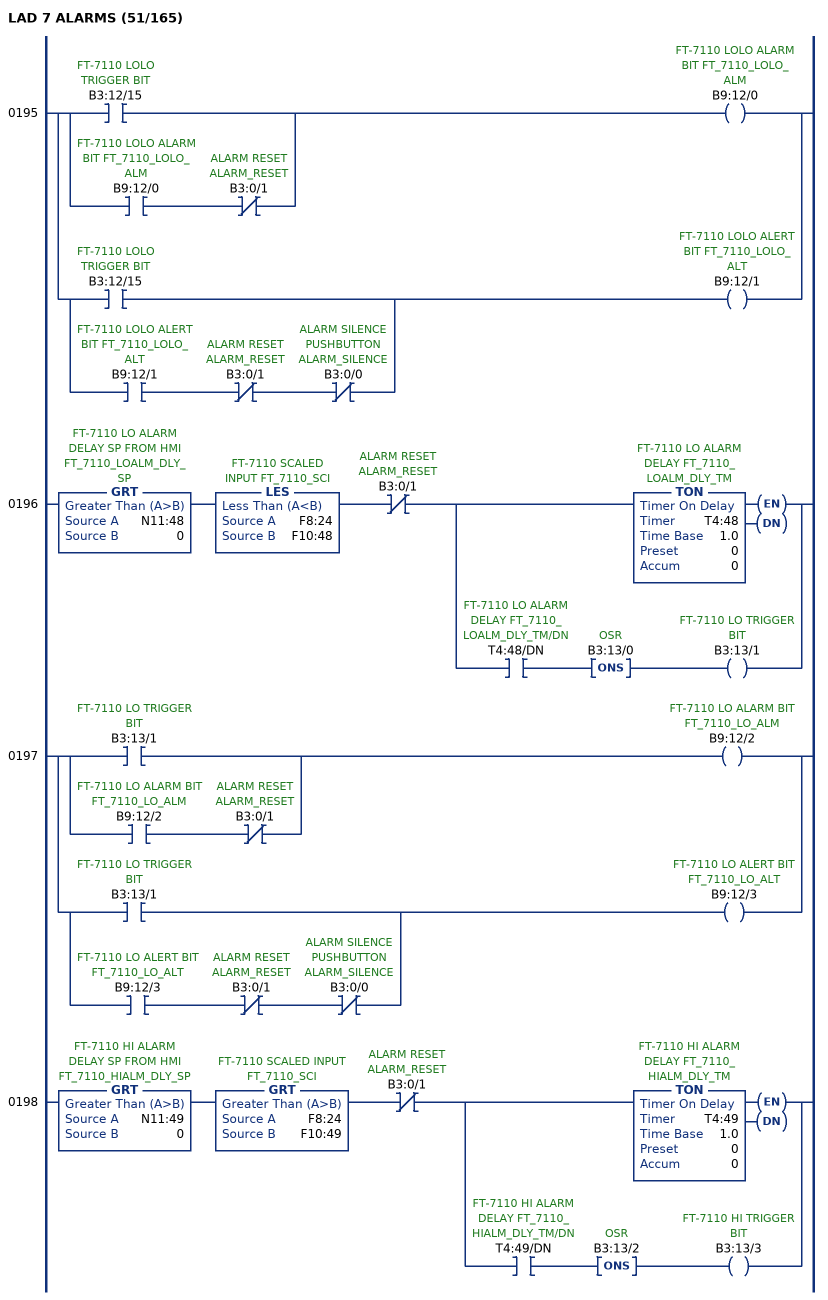
% Rung: 195 %
SOR BST BST XIC B3:12/15 NXB XIC B9:12/0 XIO B3:0/1 BND OTE B9:12/0 NXB BST XIC B3:12/15 NXB XIC B9:12/1 XIO B3:0/1 XIO B3:0/0 BND OTE B9:12/1 BND EOR
%   B3:12/15  "FT-7110 LOLO TRIGGER BIT" %
%   B9:12/0  FT_7110_LOLO_ALM  "FT-7110 LOLO ALARM BIT" %
%   B3:0/1  ALARM_RESET  "ALARM RESET" %
%   B9:12/1  FT_7110_LOLO_ALT  "FT-7110 LOLO ALERT BIT" %
%   B3:0/0  ALARM_SILENCE  "ALARM SILENCE PUSHBUTTON" %
% Rung: 196 %
SOR GRT N11:48 0 LES F8:24 F10:48 XIO B3:0/1 BST TON T4:48 1.0 0 0 NXB XIC T4:48/DN OSR B3:13/0 OTE B3:13/1 BND EOR
%   N11:48  FT_7110_LOALM_DLY_SP  "FT-7110 LO ALARM DELAY SP FROM HMI" %
%   F8:24  FT_7110_SCI  "FT-7110 SCALED INPUT" %
%   F10:48  FT_7110_LOALM_SP  "FT-7110 LO ALARM SP" %
%   B3:0/1  ALARM_RESET  "ALARM RESET" %
%   T4:48  FT_7110_LOALM_DLY_TM  "FT-7110 LO ALARM DELAY" %
%   B3:13/0  "OSR" %
%   B3:13/1  "FT-7110 LO TRIGGER BIT" %
% Rung: 197 %
SOR BST BST XIC B3:13/1 NXB XIC B9:12/2 XIO B3:0/1 BND OTE B9:12/2 NXB BST XIC B3:13/1 NXB XIC B9:12/3 XIO B3:0/1 XIO B3:0/0 BND OTE B9:12/3 BND EOR
%   B3:13/1  "FT-7110 LO TRIGGER BIT" %
%   B9:12/2  FT_7110_LO_ALM  "FT-7110 LO ALARM BIT" %
%   B3:0/1  ALARM_RESET  "ALARM RESET" %
%   B9:12/3  FT_7110_LO_ALT  "FT-7110 LO ALERT BIT" %
%   B3:0/0  ALARM_SILENCE  "ALARM SILENCE PUSHBUTTON" %
% Rung: 198 %
SOR GRT N11:49 0 GRT F8:24 F10:49 XIO B3:0/1 BST TON T4:49 1.0 0 0 NXB XIC T4:49/DN OSR B3:13/2 OTE B3:13/3 BND EOR
%   N11:49  FT_7110_HIALM_DLY_SP  "FT-7110 HI ALARM DELAY SP FROM HMI" %
%   F8:24  FT_7110_SCI  "FT-7110 SCALED INPUT" %
%   F10:49  FT_7110_HIALM_SP  "FT-7110 HI ALARM SP" %
%   B3:0/1  ALARM_RESET  "ALARM RESET" %
%   T4:49  FT_7110_HIALM_DLY_TM  "FT-7110 HI ALARM DELAY" %
%   B3:13/2  "OSR" %
%   B3:13/3  "FT-7110 HI TRIGGER BIT" %

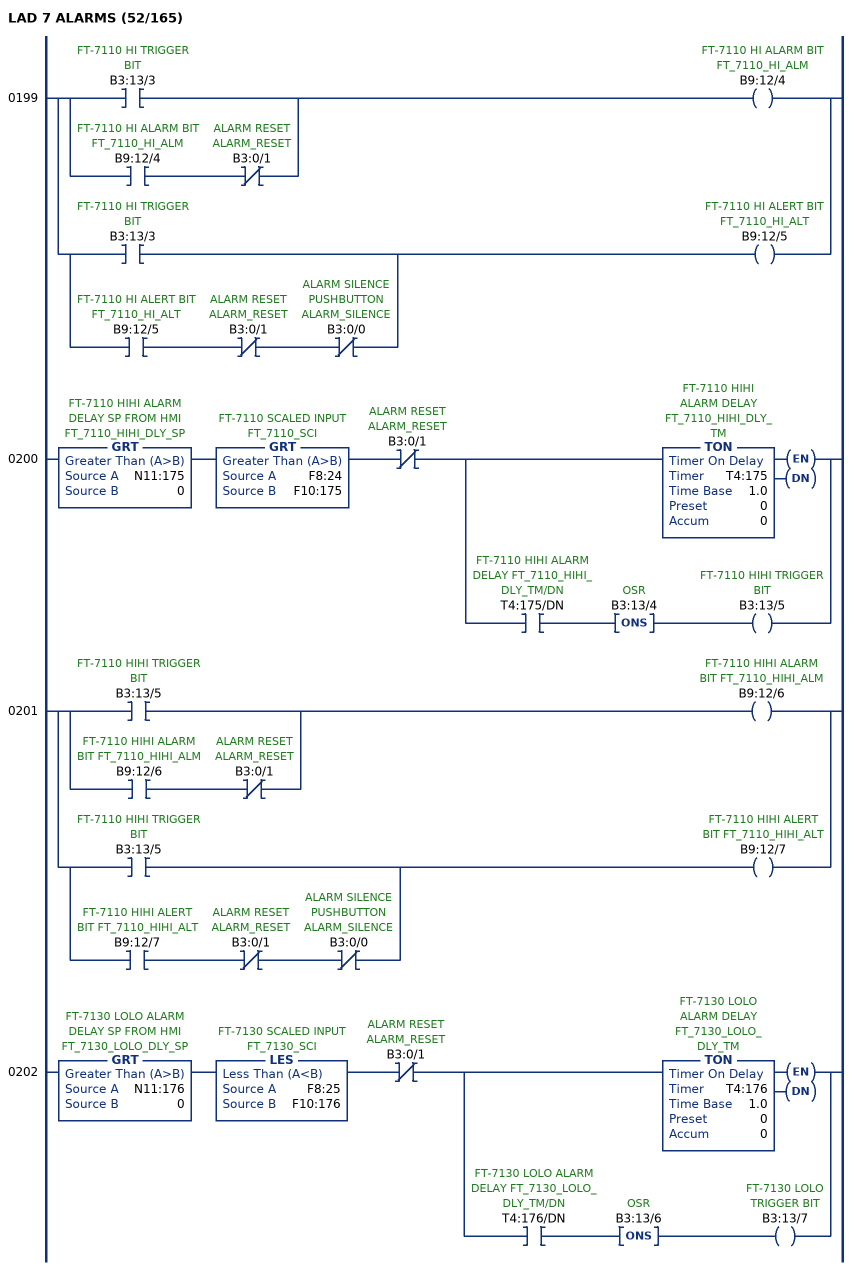
% Rung: 199 %
SOR BST BST XIC B3:13/3 NXB XIC B9:12/4 XIO B3:0/1 BND OTE B9:12/4 NXB BST XIC B3:13/3 NXB XIC B9:12/5 XIO B3:0/1 XIO B3:0/0 BND OTE B9:12/5 BND EOR
%   B3:13/3  "FT-7110 HI TRIGGER BIT" %
%   B9:12/4  FT_7110_HI_ALM  "FT-7110 HI ALARM BIT" %
%   B3:0/1  ALARM_RESET  "ALARM RESET" %
%   B9:12/5  FT_7110_HI_ALT  "FT-7110 HI ALERT BIT" %
%   B3:0/0  ALARM_SILENCE  "ALARM SILENCE PUSHBUTTON" %
% Rung: 200 %
SOR GRT N11:175 0 GRT F8:24 F10:175 XIO B3:0/1 BST TON T4:175 1.0 0 0 NXB XIC T4:175/DN OSR B3:13/4 OTE B3:13/5 BND EOR
%   N11:175  FT_7110_HIHI_DLY_SP  "FT-7110 HIHI ALARM DELAY SP FROM HMI" %
%   F8:24  FT_7110_SCI  "FT-7110 SCALED INPUT" %
%   F10:175  FT_7110_HIHI_SP  "FT-7110 HIHI ALARM SP" %
%   B3:0/1  ALARM_RESET  "ALARM RESET" %
%   T4:175  FT_7110_HIHI_DLY_TM  "FT-7110 HIHI ALARM DELAY" %
%   B3:13/4  "OSR" %
%   B3:13/5  "FT-7110 HIHI TRIGGER BIT" %
% Rung: 201 %
SOR BST BST XIC B3:13/5 NXB XIC B9:12/6 XIO B3:0/1 BND OTE B9:12/6 NXB BST XIC B3:13/5 NXB XIC B9:12/7 XIO B3:0/1 XIO B3:0/0 BND OTE B9:12/7 BND EOR
%   B3:13/5  "FT-7110 HIHI TRIGGER BIT" %
%   B9:12/6  FT_7110_HIHI_ALM  "FT-7110 HIHI ALARM BIT" %
%   B3:0/1  ALARM_RESET  "ALARM RESET" %
%   B9:12/7  FT_7110_HIHI_ALT  "FT-7110 HIHI ALERT BIT" %
%   B3:0/0  ALARM_SILENCE  "ALARM SILENCE PUSHBUTTON" %
% Rung: 202 %
SOR GRT N11:176 0 LES F8:25 F10:176 XIO B3:0/1 BST TON T4:176 1.0 0 0 NXB XIC T4:176/DN OSR B3:13/6 OTE B3:13/7 BND EOR
%   N11:176  FT_7130_LOLO_DLY_SP  "FT-7130 LOLO ALARM DELAY SP FROM HMI" %
%   F8:25  FT_7130_SCI  "FT-7130 SCALED INPUT" %
%   F10:176  FT_7130_LOLO_SP  "FT-7130 LOLO ALARM SP" %
%   B3:0/1  ALARM_RESET  "ALARM RESET" %
%   T4:176  FT_7130_LOLO_DLY_TM  "FT-7130 LOLO ALARM DELAY" %
%   B3:13/6  "OSR" %
%   B3:13/7  "FT-7130 LOLO TRIGGER BIT" %

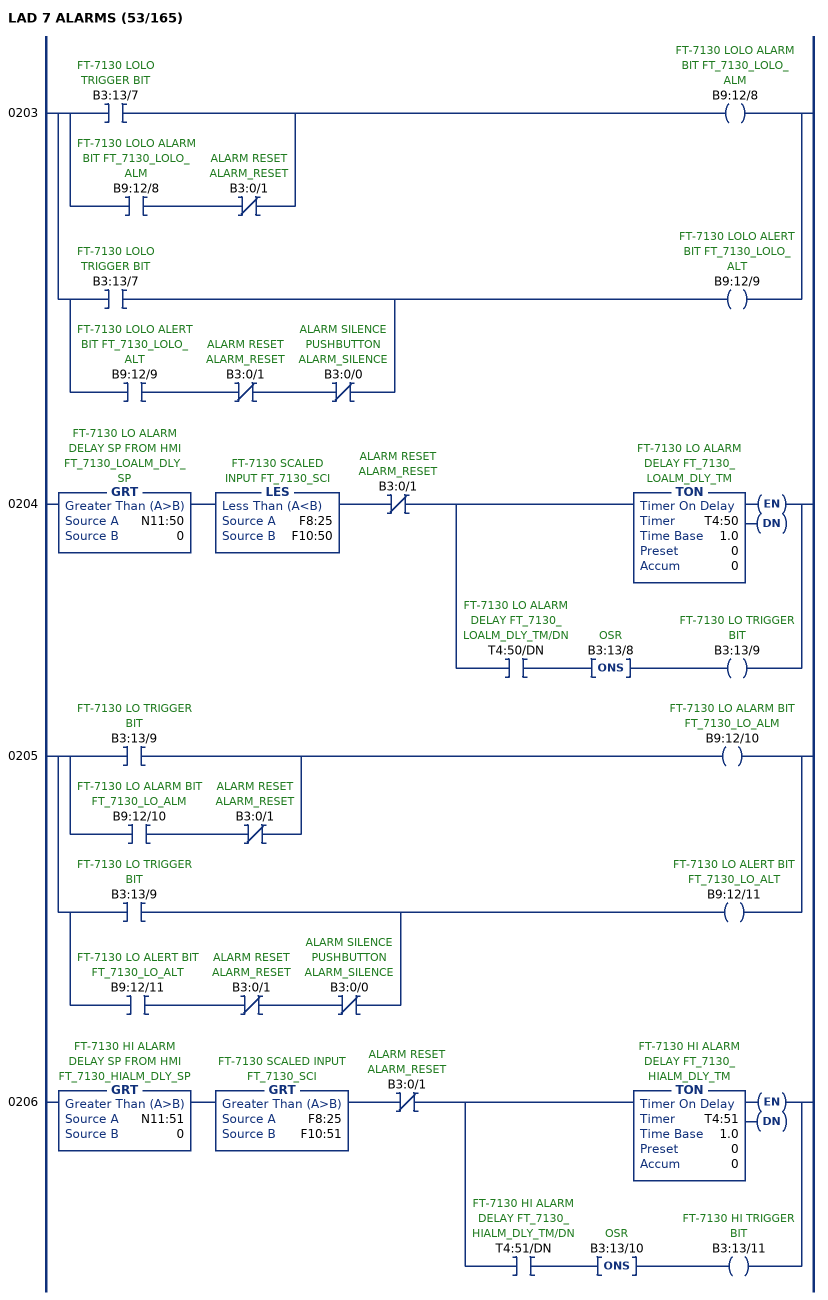
% Rung: 203 %
SOR BST BST XIC B3:13/7 NXB XIC B9:12/8 XIO B3:0/1 BND OTE B9:12/8 NXB BST XIC B3:13/7 NXB XIC B9:12/9 XIO B3:0/1 XIO B3:0/0 BND OTE B9:12/9 BND EOR
%   B3:13/7  "FT-7130 LOLO TRIGGER BIT" %
%   B9:12/8  FT_7130_LOLO_ALM  "FT-7130 LOLO ALARM BIT" %
%   B3:0/1  ALARM_RESET  "ALARM RESET" %
%   B9:12/9  FT_7130_LOLO_ALT  "FT-7130 LOLO ALERT BIT" %
%   B3:0/0  ALARM_SILENCE  "ALARM SILENCE PUSHBUTTON" %
% Rung: 204 %
SOR GRT N11:50 0 LES F8:25 F10:50 XIO B3:0/1 BST TON T4:50 1.0 0 0 NXB XIC T4:50/DN OSR B3:13/8 OTE B3:13/9 BND EOR
%   N11:50  FT_7130_LOALM_DLY_SP  "FT-7130 LO ALARM DELAY SP FROM HMI" %
%   F8:25  FT_7130_SCI  "FT-7130 SCALED INPUT" %
%   F10:50  FT_7130_LOALM_SP  "FT-7130 LO ALARM SP" %
%   B3:0/1  ALARM_RESET  "ALARM RESET" %
%   T4:50  FT_7130_LOALM_DLY_TM  "FT-7130 LO ALARM DELAY" %
%   B3:13/8  "OSR" %
%   B3:13/9  "FT-7130 LO TRIGGER BIT" %
% Rung: 205 %
SOR BST BST XIC B3:13/9 NXB XIC B9:12/10 XIO B3:0/1 BND OTE B9:12/10 NXB BST XIC B3:13/9 NXB XIC B9:12/11 XIO B3:0/1 XIO B3:0/0 BND OTE B9:12/11 BND EOR
%   B3:13/9  "FT-7130 LO TRIGGER BIT" %
%   B9:12/10  FT_7130_LO_ALM  "FT-7130 LO ALARM BIT" %
%   B3:0/1  ALARM_RESET  "ALARM RESET" %
%   B9:12/11  FT_7130_LO_ALT  "FT-7130 LO ALERT BIT" %
%   B3:0/0  ALARM_SILENCE  "ALARM SILENCE PUSHBUTTON" %
% Rung: 206 %
SOR GRT N11:51 0 GRT F8:25 F10:51 XIO B3:0/1 BST TON T4:51 1.0 0 0 NXB XIC T4:51/DN OSR B3:13/10 OTE B3:13/11 BND EOR
%   N11:51  FT_7130_HIALM_DLY_SP  "FT-7130 HI ALARM DELAY SP FROM HMI" %
%   F8:25  FT_7130_SCI  "FT-7130 SCALED INPUT" %
%   F10:51  FT_7130_HIALM_SP  "FT-7130 HI ALARM SP" %
%   B3:0/1  ALARM_RESET  "ALARM RESET" %
%   T4:51  FT_7130_HIALM_DLY_TM  "FT-7130 HI ALARM DELAY" %
%   B3:13/10  "OSR" %
%   B3:13/11  "FT-7130 HI TRIGGER BIT" %

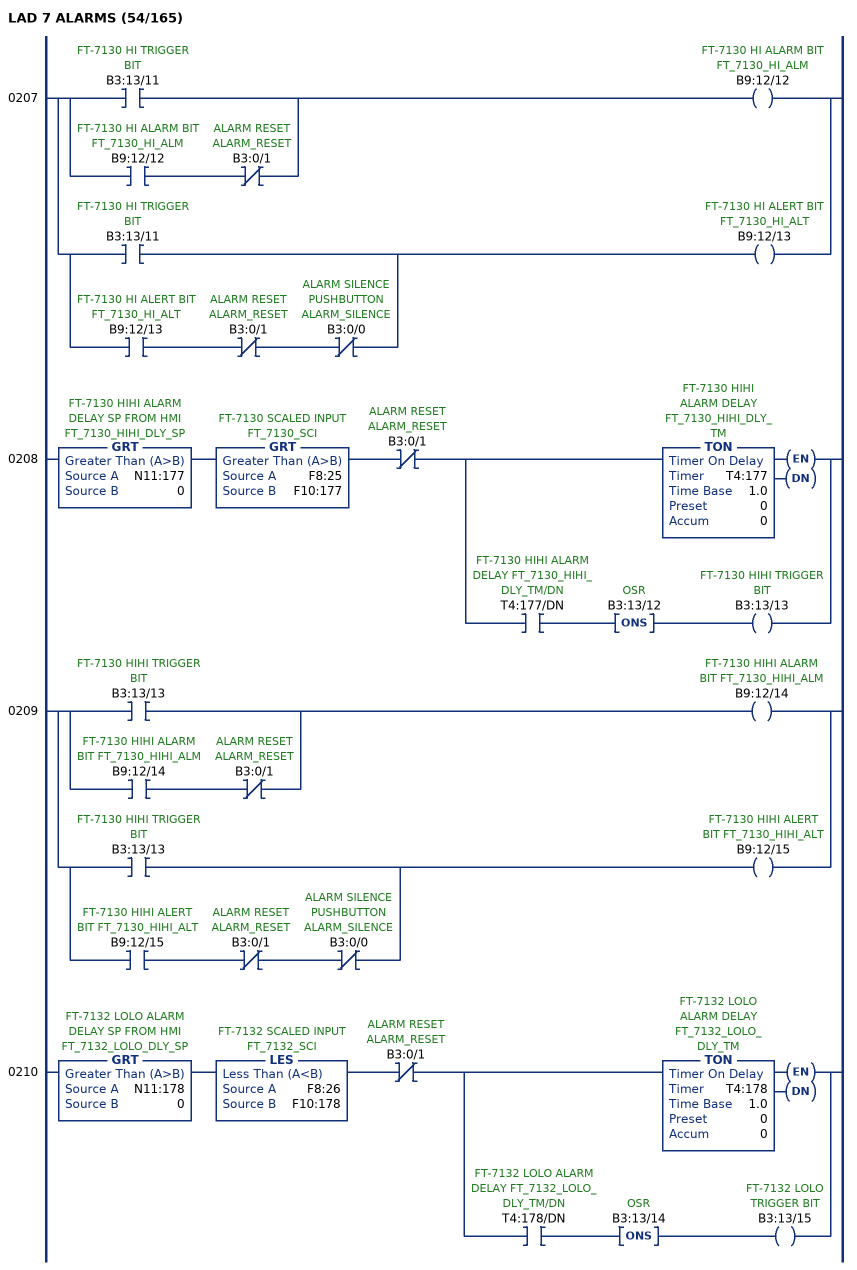
% Rung: 207 %
SOR BST BST XIC B3:13/11 NXB XIC B9:12/12 XIO B3:0/1 BND OTE B9:12/12 NXB BST XIC B3:13/11 NXB XIC B9:12/13 XIO B3:0/1 XIO B3:0/0 BND OTE B9:12/13 BND EOR
%   B3:13/11  "FT-7130 HI TRIGGER BIT" %
%   B9:12/12  FT_7130_HI_ALM  "FT-7130 HI ALARM BIT" %
%   B3:0/1  ALARM_RESET  "ALARM RESET" %
%   B9:12/13  FT_7130_HI_ALT  "FT-7130 HI ALERT BIT" %
%   B3:0/0  ALARM_SILENCE  "ALARM SILENCE PUSHBUTTON" %
% Rung: 208 %
SOR GRT N11:177 0 GRT F8:25 F10:177 XIO B3:0/1 BST TON T4:177 1.0 0 0 NXB XIC T4:177/DN OSR B3:13/12 OTE B3:13/13 BND EOR
%   N11:177  FT_7130_HIHI_DLY_SP  "FT-7130 HIHI ALARM DELAY SP FROM HMI" %
%   F8:25  FT_7130_SCI  "FT-7130 SCALED INPUT" %
%   F10:177  FT_7130_HIHI_SP  "FT-7130 HIHI ALARM SP" %
%   B3:0/1  ALARM_RESET  "ALARM RESET" %
%   T4:177  FT_7130_HIHI_DLY_TM  "FT-7130 HIHI ALARM DELAY" %
%   B3:13/12  "OSR" %
%   B3:13/13  "FT-7130 HIHI TRIGGER BIT" %
% Rung: 209 %
SOR BST BST XIC B3:13/13 NXB XIC B9:12/14 XIO B3:0/1 BND OTE B9:12/14 NXB BST XIC B3:13/13 NXB XIC B9:12/15 XIO B3:0/1 XIO B3:0/0 BND OTE B9:12/15 BND EOR
%   B3:13/13  "FT-7130 HIHI TRIGGER BIT" %
%   B9:12/14  FT_7130_HIHI_ALM  "FT-7130 HIHI ALARM BIT" %
%   B3:0/1  ALARM_RESET  "ALARM RESET" %
%   B9:12/15  FT_7130_HIHI_ALT  "FT-7130 HIHI ALERT BIT" %
%   B3:0/0  ALARM_SILENCE  "ALARM SILENCE PUSHBUTTON" %
% Rung: 210 %
SOR GRT N11:178 0 LES F8:26 F10:178 XIO B3:0/1 BST TON T4:178 1.0 0 0 NXB XIC T4:178/DN OSR B3:13/14 OTE B3:13/15 BND EOR
%   N11:178  FT_7132_LOLO_DLY_SP  "FT-7132 LOLO ALARM DELAY SP FROM HMI" %
%   F8:26  FT_7132_SCI  "FT-7132 SCALED INPUT" %
%   F10:178  FT_7132_LOLO_SP  "FT-7132 LOLO ALARM SP" %
%   B3:0/1  ALARM_RESET  "ALARM RESET" %
%   T4:178  FT_7132_LOLO_DLY_TM  "FT-7132 LOLO ALARM DELAY" %
%   B3:13/14  "OSR" %
%   B3:13/15  "FT-7132 LOLO TRIGGER BIT" %

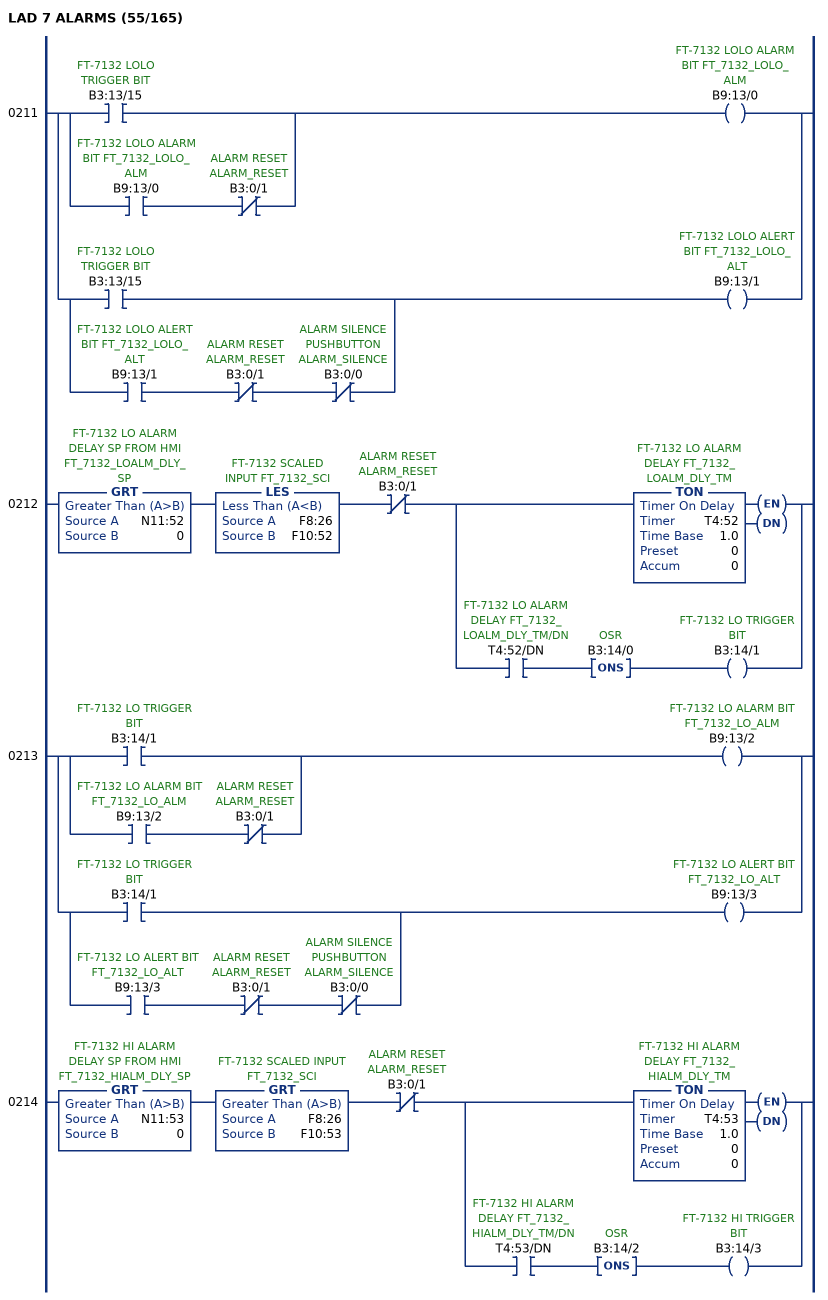
% Rung: 211 %
SOR BST BST XIC B3:13/15 NXB XIC B9:13/0 XIO B3:0/1 BND OTE B9:13/0 NXB BST XIC B3:13/15 NXB XIC B9:13/1 XIO B3:0/1 XIO B3:0/0 BND OTE B9:13/1 BND EOR
%   B3:13/15  "FT-7132 LOLO TRIGGER BIT" %
%   B9:13/0  FT_7132_LOLO_ALM  "FT-7132 LOLO ALARM BIT" %
%   B3:0/1  ALARM_RESET  "ALARM RESET" %
%   B9:13/1  FT_7132_LOLO_ALT  "FT-7132 LOLO ALERT BIT" %
%   B3:0/0  ALARM_SILENCE  "ALARM SILENCE PUSHBUTTON" %
% Rung: 212 %
SOR GRT N11:52 0 LES F8:26 F10:52 XIO B3:0/1 BST TON T4:52 1.0 0 0 NXB XIC T4:52/DN OSR B3:14/0 OTE B3:14/1 BND EOR
%   N11:52  FT_7132_LOALM_DLY_SP  "FT-7132 LO ALARM DELAY SP FROM HMI" %
%   F8:26  FT_7132_SCI  "FT-7132 SCALED INPUT" %
%   F10:52  FT_7132_LOALM_SP  "FT-7132 LO ALARM SP" %
%   B3:0/1  ALARM_RESET  "ALARM RESET" %
%   T4:52  FT_7132_LOALM_DLY_TM  "FT-7132 LO ALARM DELAY" %
%   B3:14/0  "OSR" %
%   B3:14/1  "FT-7132 LO TRIGGER BIT" %
% Rung: 213 %
SOR BST BST XIC B3:14/1 NXB XIC B9:13/2 XIO B3:0/1 BND OTE B9:13/2 NXB BST XIC B3:14/1 NXB XIC B9:13/3 XIO B3:0/1 XIO B3:0/0 BND OTE B9:13/3 BND EOR
%   B3:14/1  "FT-7132 LO TRIGGER BIT" %
%   B9:13/2  FT_7132_LO_ALM  "FT-7132 LO ALARM BIT" %
%   B3:0/1  ALARM_RESET  "ALARM RESET" %
%   B9:13/3  FT_7132_LO_ALT  "FT-7132 LO ALERT BIT" %
%   B3:0/0  ALARM_SILENCE  "ALARM SILENCE PUSHBUTTON" %
% Rung: 214 %
SOR GRT N11:53 0 GRT F8:26 F10:53 XIO B3:0/1 BST TON T4:53 1.0 0 0 NXB XIC T4:53/DN OSR B3:14/2 OTE B3:14/3 BND EOR
%   N11:53  FT_7132_HIALM_DLY_SP  "FT-7132 HI ALARM DELAY SP FROM HMI" %
%   F8:26  FT_7132_SCI  "FT-7132 SCALED INPUT" %
%   F10:53  FT_7132_HIALM_SP  "FT-7132 HI ALARM SP" %
%   B3:0/1  ALARM_RESET  "ALARM RESET" %
%   T4:53  FT_7132_HIALM_DLY_TM  "FT-7132 HI ALARM DELAY" %
%   B3:14/2  "OSR" %
%   B3:14/3  "FT-7132 HI TRIGGER BIT" %

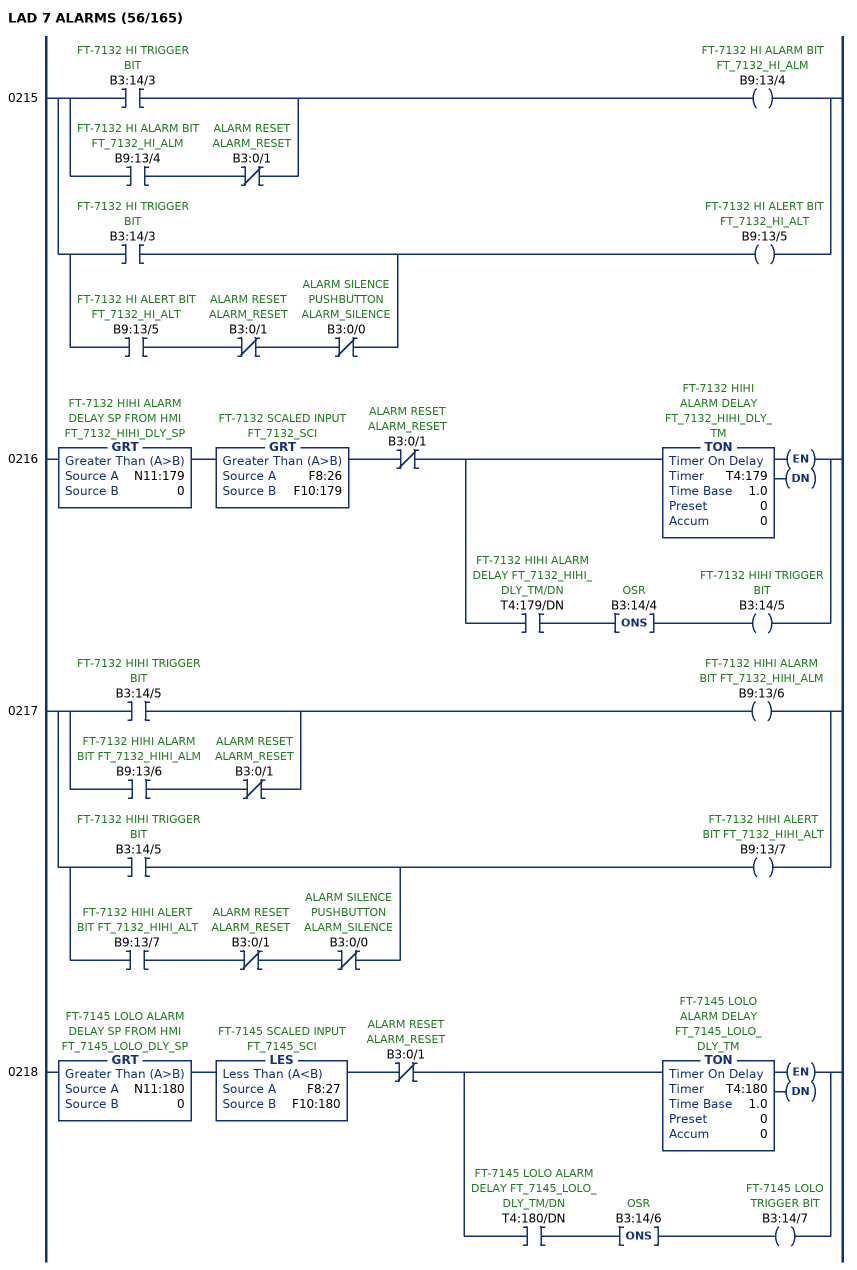
% Rung: 215 %
SOR BST BST XIC B3:14/3 NXB XIC B9:13/4 XIO B3:0/1 BND OTE B9:13/4 NXB BST XIC B3:14/3 NXB XIC B9:13/5 XIO B3:0/1 XIO B3:0/0 BND OTE B9:13/5 BND EOR
%   B3:14/3  "FT-7132 HI TRIGGER BIT" %
%   B9:13/4  FT_7132_HI_ALM  "FT-7132 HI ALARM BIT" %
%   B3:0/1  ALARM_RESET  "ALARM RESET" %
%   B9:13/5  FT_7132_HI_ALT  "FT-7132 HI ALERT BIT" %
%   B3:0/0  ALARM_SILENCE  "ALARM SILENCE PUSHBUTTON" %
% Rung: 216 %
SOR GRT N11:179 0 GRT F8:26 F10:179 XIO B3:0/1 BST TON T4:179 1.0 0 0 NXB XIC T4:179/DN OSR B3:14/4 OTE B3:14/5 BND EOR
%   N11:179  FT_7132_HIHI_DLY_SP  "FT-7132 HIHI ALARM DELAY SP FROM HMI" %
%   F8:26  FT_7132_SCI  "FT-7132 SCALED INPUT" %
%   F10:179  FT_7132_HIHI_SP  "FT-7132 HIHI ALARM SP" %
%   B3:0/1  ALARM_RESET  "ALARM RESET" %
%   T4:179  FT_7132_HIHI_DLY_TM  "FT-7132 HIHI ALARM DELAY" %
%   B3:14/4  "OSR" %
%   B3:14/5  "FT-7132 HIHI TRIGGER BIT" %
% Rung: 217 %
SOR BST BST XIC B3:14/5 NXB XIC B9:13/6 XIO B3:0/1 BND OTE B9:13/6 NXB BST XIC B3:14/5 NXB XIC B9:13/7 XIO B3:0/1 XIO B3:0/0 BND OTE B9:13/7 BND EOR
%   B3:14/5  "FT-7132 HIHI TRIGGER BIT" %
%   B9:13/6  FT_7132_HIHI_ALM  "FT-7132 HIHI ALARM BIT" %
%   B3:0/1  ALARM_RESET  "ALARM RESET" %
%   B9:13/7  FT_7132_HIHI_ALT  "FT-7132 HIHI ALERT BIT" %
%   B3:0/0  ALARM_SILENCE  "ALARM SILENCE PUSHBUTTON" %
% Rung: 218 %
SOR GRT N11:180 0 LES F8:27 F10:180 XIO B3:0/1 BST TON T4:180 1.0 0 0 NXB XIC T4:180/DN OSR B3:14/6 OTE B3:14/7 BND EOR
%   N11:180  FT_7145_LOLO_DLY_SP  "FT-7145 LOLO ALARM DELAY SP FROM HMI" %
%   F8:27  FT_7145_SCI  "FT-7145 SCALED INPUT" %
%   F10:180  FT_7145_LOLO_SP  "FT-7145 LOLO ALARM SP" %
%   B3:0/1  ALARM_RESET  "ALARM RESET" %
%   T4:180  FT_7145_LOLO_DLY_TM  "FT-7145 LOLO ALARM DELAY" %
%   B3:14/6  "OSR" %
%   B3:14/7  "FT-7145 LOLO TRIGGER BIT" %

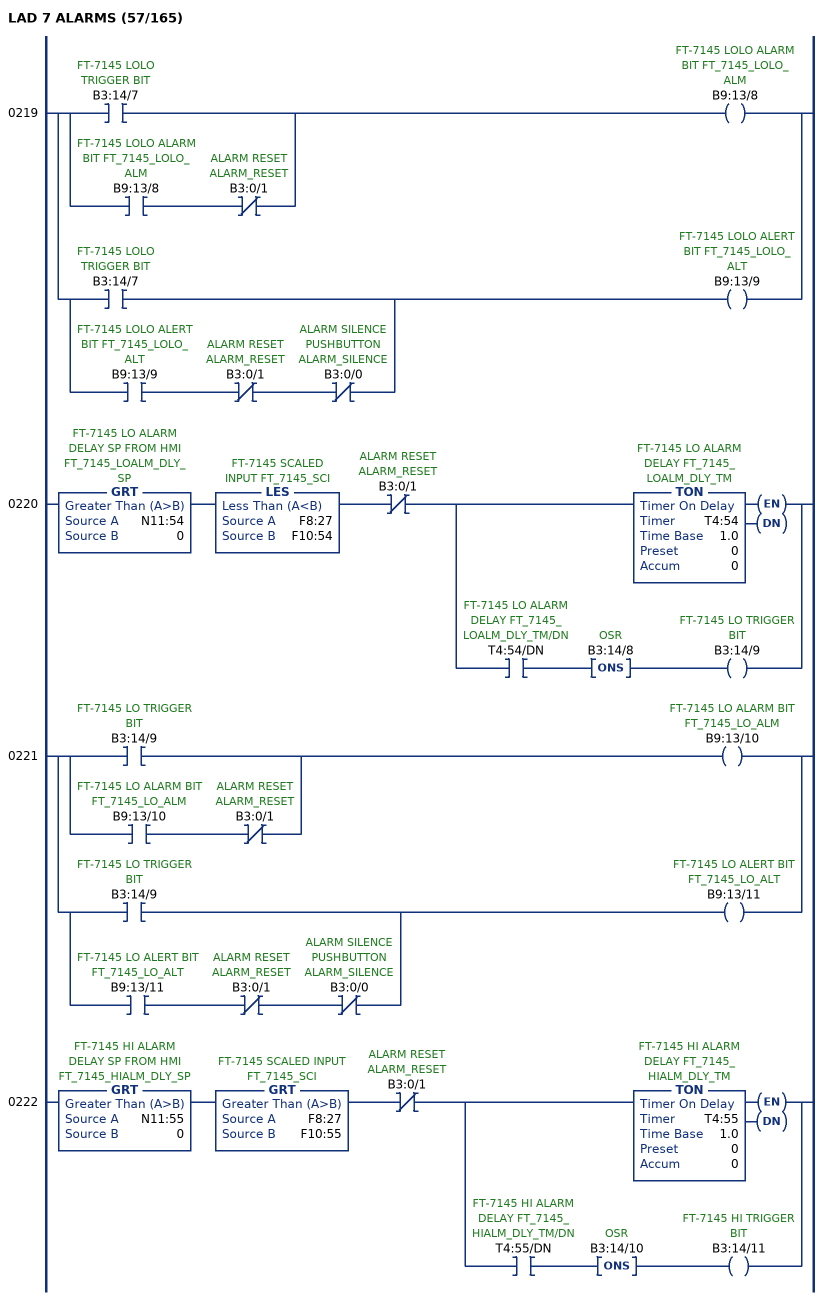
% Rung: 219 %
SOR BST BST XIC B3:14/7 NXB XIC B9:13/8 XIO B3:0/1 BND OTE B9:13/8 NXB BST XIC B3:14/7 NXB XIC B9:13/9 XIO B3:0/1 XIO B3:0/0 BND OTE B9:13/9 BND EOR
%   B3:14/7  "FT-7145 LOLO TRIGGER BIT" %
%   B9:13/8  FT_7145_LOLO_ALM  "FT-7145 LOLO ALARM BIT" %
%   B3:0/1  ALARM_RESET  "ALARM RESET" %
%   B9:13/9  FT_7145_LOLO_ALT  "FT-7145 LOLO ALERT BIT" %
%   B3:0/0  ALARM_SILENCE  "ALARM SILENCE PUSHBUTTON" %
% Rung: 220 %
SOR GRT N11:54 0 LES F8:27 F10:54 XIO B3:0/1 BST TON T4:54 1.0 0 0 NXB XIC T4:54/DN OSR B3:14/8 OTE B3:14/9 BND EOR
%   N11:54  FT_7145_LOALM_DLY_SP  "FT-7145 LO ALARM DELAY SP FROM HMI" %
%   F8:27  FT_7145_SCI  "FT-7145 SCALED INPUT" %
%   F10:54  FT_7145_LOALM_SP  "FT-7145 LO ALARM SP" %
%   B3:0/1  ALARM_RESET  "ALARM RESET" %
%   T4:54  FT_7145_LOALM_DLY_TM  "FT-7145 LO ALARM DELAY" %
%   B3:14/8  "OSR" %
%   B3:14/9  "FT-7145 LO TRIGGER BIT" %
% Rung: 221 %
SOR BST BST XIC B3:14/9 NXB XIC B9:13/10 XIO B3:0/1 BND OTE B9:13/10 NXB BST XIC B3:14/9 NXB XIC B9:13/11 XIO B3:0/1 XIO B3:0/0 BND OTE B9:13/11 BND EOR
%   B3:14/9  "FT-7145 LO TRIGGER BIT" %
%   B9:13/10  FT_7145_LO_ALM  "FT-7145 LO ALARM BIT" %
%   B3:0/1  ALARM_RESET  "ALARM RESET" %
%   B9:13/11  FT_7145_LO_ALT  "FT-7145 LO ALERT BIT" %
%   B3:0/0  ALARM_SILENCE  "ALARM SILENCE PUSHBUTTON" %
% Rung: 222 %
SOR GRT N11:55 0 GRT F8:27 F10:55 XIO B3:0/1 BST TON T4:55 1.0 0 0 NXB XIC T4:55/DN OSR B3:14/10 OTE B3:14/11 BND EOR
%   N11:55  FT_7145_HIALM_DLY_SP  "FT-7145 HI ALARM DELAY SP FROM HMI" %
%   F8:27  FT_7145_SCI  "FT-7145 SCALED INPUT" %
%   F10:55  FT_7145_HIALM_SP  "FT-7145 HI ALARM SP" %
%   B3:0/1  ALARM_RESET  "ALARM RESET" %
%   T4:55  FT_7145_HIALM_DLY_TM  "FT-7145 HI ALARM DELAY" %
%   B3:14/10  "OSR" %
%   B3:14/11  "FT-7145 HI TRIGGER BIT" %

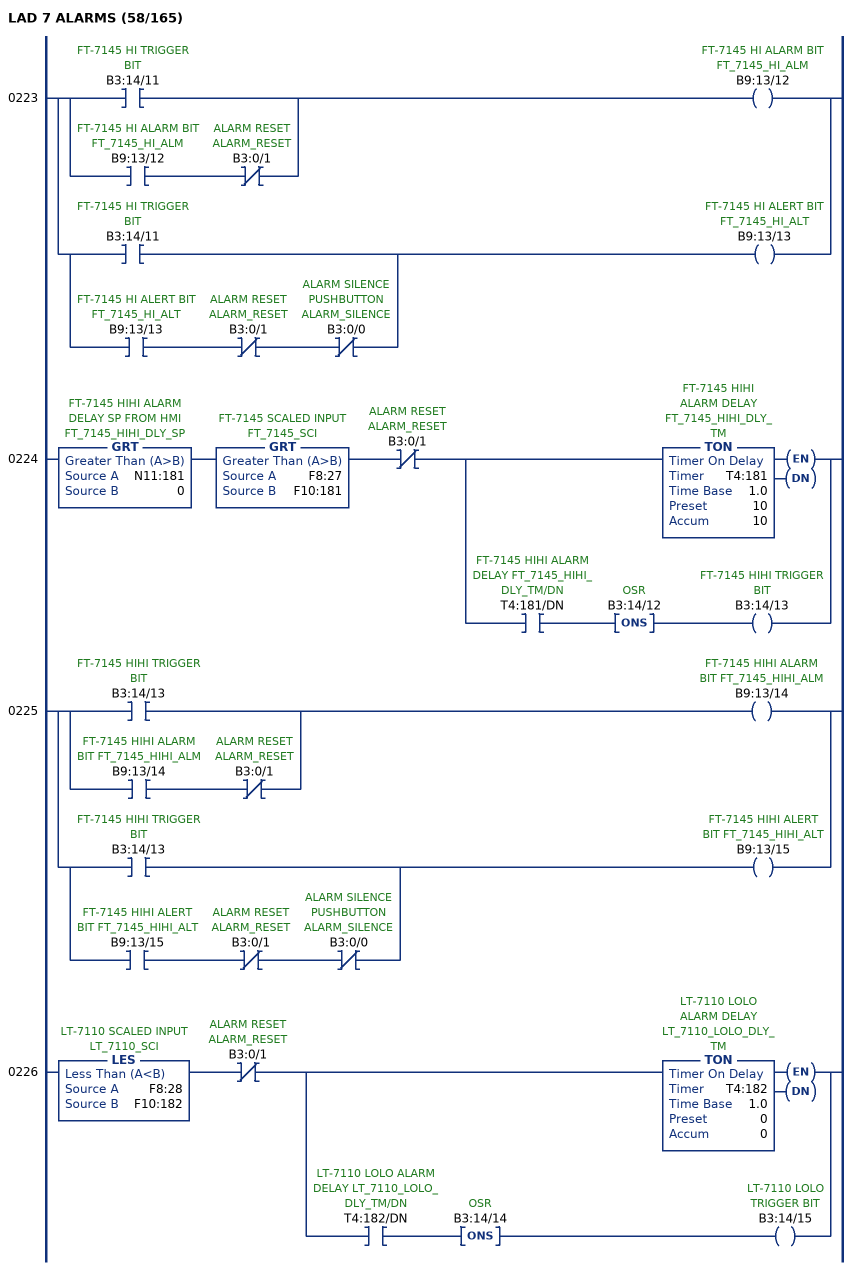
% Rung: 223 %
SOR BST BST XIC B3:14/11 NXB XIC B9:13/12 XIO B3:0/1 BND OTE B9:13/12 NXB BST XIC B3:14/11 NXB XIC B9:13/13 XIO B3:0/1 XIO B3:0/0 BND OTE B9:13/13 BND EOR
%   B3:14/11  "FT-7145 HI TRIGGER BIT" %
%   B9:13/12  FT_7145_HI_ALM  "FT-7145 HI ALARM BIT" %
%   B3:0/1  ALARM_RESET  "ALARM RESET" %
%   B9:13/13  FT_7145_HI_ALT  "FT-7145 HI ALERT BIT" %
%   B3:0/0  ALARM_SILENCE  "ALARM SILENCE PUSHBUTTON" %
% Rung: 224 %
SOR GRT N11:181 0 GRT F8:27 F10:181 XIO B3:0/1 BST TON T4:181 1.0 10 10 NXB XIC T4:181/DN OSR B3:14/12 OTE B3:14/13 BND EOR
%   N11:181  FT_7145_HIHI_DLY_SP  "FT-7145 HIHI ALARM DELAY SP FROM HMI" %
%   F8:27  FT_7145_SCI  "FT-7145 SCALED INPUT" %
%   F10:181  FT_7145_HIHI_SP  "FT-7145 HIHI ALARM SP" %
%   B3:0/1  ALARM_RESET  "ALARM RESET" %
%   T4:181  FT_7145_HIHI_DLY_TM  "FT-7145 HIHI ALARM DELAY" %
%   B3:14/12  "OSR" %
%   B3:14/13  "FT-7145 HIHI TRIGGER BIT" %
% Rung: 225 %
SOR BST BST XIC B3:14/13 NXB XIC B9:13/14 XIO B3:0/1 BND OTE B9:13/14 NXB BST XIC B3:14/13 NXB XIC B9:13/15 XIO B3:0/1 XIO B3:0/0 BND OTE B9:13/15 BND EOR
%   B3:14/13  "FT-7145 HIHI TRIGGER BIT" %
%   B9:13/14  FT_7145_HIHI_ALM  "FT-7145 HIHI ALARM BIT" %
%   B3:0/1  ALARM_RESET  "ALARM RESET" %
%   B9:13/15  FT_7145_HIHI_ALT  "FT-7145 HIHI ALERT BIT" %
%   B3:0/0  ALARM_SILENCE  "ALARM SILENCE PUSHBUTTON" %
% Rung: 226 %
SOR LES F8:28 F10:182 XIO B3:0/1 BST TON T4:182 1.0 0 0 NXB XIC T4:182/DN OSR B3:14/14 OTE B3:14/15 BND EOR
%   F8:28  LT_7110_SCI  "LT-7110 SCALED INPUT" %
%   F10:182  LT_7110_LOLO_SP  "LT-7110 LOLO ALARM SP" %
%   B3:0/1  ALARM_RESET  "ALARM RESET" %
%   T4:182  LT_7110_LOLO_DLY_TM  "LT-7110 LOLO ALARM DELAY" %
%   B3:14/14  "OSR" %
%   B3:14/15  "LT-7110 LOLO TRIGGER BIT" %

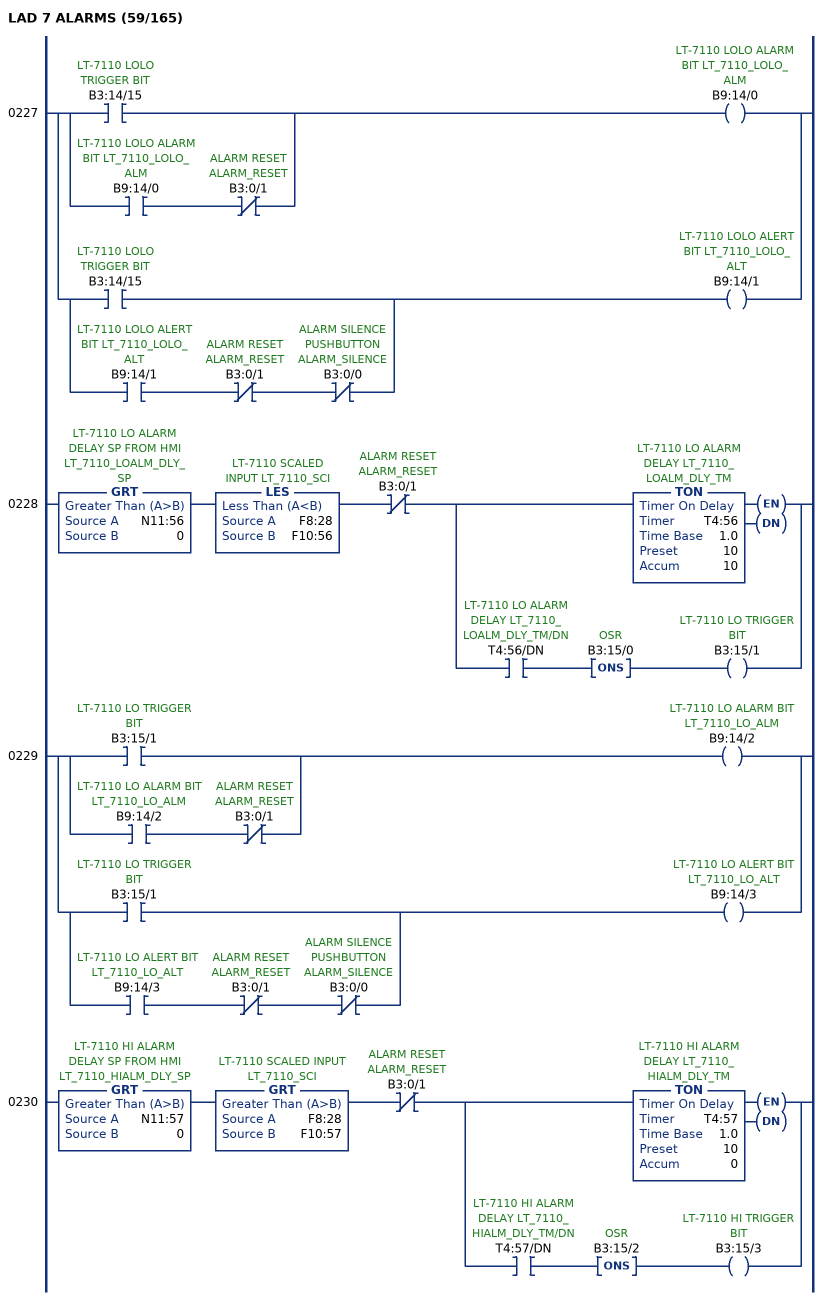
% Rung: 227 %
SOR BST BST XIC B3:14/15 NXB XIC B9:14/0 XIO B3:0/1 BND OTE B9:14/0 NXB BST XIC B3:14/15 NXB XIC B9:14/1 XIO B3:0/1 XIO B3:0/0 BND OTE B9:14/1 BND EOR
%   B3:14/15  "LT-7110 LOLO TRIGGER BIT" %
%   B9:14/0  LT_7110_LOLO_ALM  "LT-7110 LOLO ALARM BIT" %
%   B3:0/1  ALARM_RESET  "ALARM RESET" %
%   B9:14/1  LT_7110_LOLO_ALT  "LT-7110 LOLO ALERT BIT" %
%   B3:0/0  ALARM_SILENCE  "ALARM SILENCE PUSHBUTTON" %
% Rung: 228 %
SOR GRT N11:56 0 LES F8:28 F10:56 XIO B3:0/1 BST TON T4:56 1.0 10 10 NXB XIC T4:56/DN OSR B3:15/0 OTE B3:15/1 BND EOR
%   N11:56  LT_7110_LOALM_DLY_SP  "LT-7110 LO ALARM DELAY SP FROM HMI" %
%   F8:28  LT_7110_SCI  "LT-7110 SCALED INPUT" %
%   F10:56  LT_7110_LOALM_SP  "LT-7110 LO ALARM SP" %
%   B3:0/1  ALARM_RESET  "ALARM RESET" %
%   T4:56  LT_7110_LOALM_DLY_TM  "LT-7110 LO ALARM DELAY" %
%   B3:15/0  "OSR" %
%   B3:15/1  "LT-7110 LO TRIGGER BIT" %
% Rung: 229 %
SOR BST BST XIC B3:15/1 NXB XIC B9:14/2 XIO B3:0/1 BND OTE B9:14/2 NXB BST XIC B3:15/1 NXB XIC B9:14/3 XIO B3:0/1 XIO B3:0/0 BND OTE B9:14/3 BND EOR
%   B3:15/1  "LT-7110 LO TRIGGER BIT" %
%   B9:14/2  LT_7110_LO_ALM  "LT-7110 LO ALARM BIT" %
%   B3:0/1  ALARM_RESET  "ALARM RESET" %
%   B9:14/3  LT_7110_LO_ALT  "LT-7110 LO ALERT BIT" %
%   B3:0/0  ALARM_SILENCE  "ALARM SILENCE PUSHBUTTON" %
% Rung: 230 %
SOR GRT N11:57 0 GRT F8:28 F10:57 XIO B3:0/1 BST TON T4:57 1.0 10 0 NXB XIC T4:57/DN OSR B3:15/2 OTE B3:15/3 BND EOR
%   N11:57  LT_7110_HIALM_DLY_SP  "LT-7110 HI ALARM DELAY SP FROM HMI" %
%   F8:28  LT_7110_SCI  "LT-7110 SCALED INPUT" %
%   F10:57  LT_7110_HIALM_SP  "LT-7110 HI ALARM SP" %
%   B3:0/1  ALARM_RESET  "ALARM RESET" %
%   T4:57  LT_7110_HIALM_DLY_TM  "LT-7110 HI ALARM DELAY" %
%   B3:15/2  "OSR" %
%   B3:15/3  "LT-7110 HI TRIGGER BIT" %

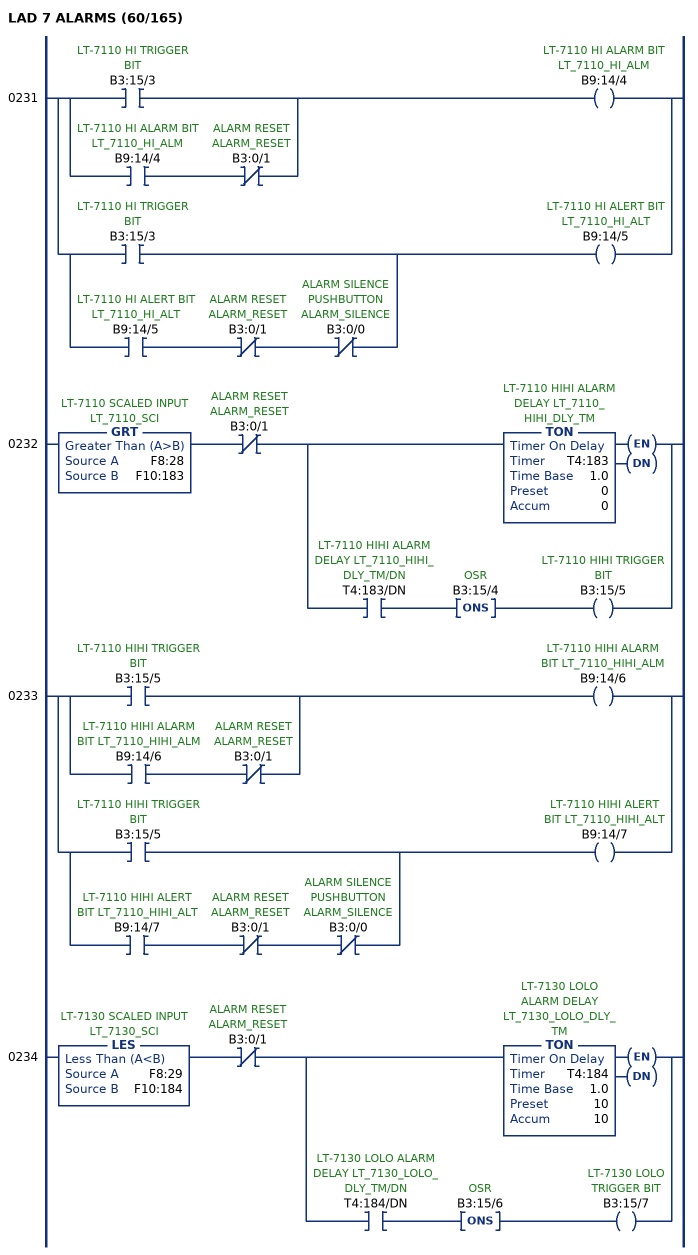
% Rung: 231 %
SOR BST BST XIC B3:15/3 NXB XIC B9:14/4 XIO B3:0/1 BND OTE B9:14/4 NXB BST XIC B3:15/3 NXB XIC B9:14/5 XIO B3:0/1 XIO B3:0/0 BND OTE B9:14/5 BND EOR
%   B3:15/3  "LT-7110 HI TRIGGER BIT" %
%   B9:14/4  LT_7110_HI_ALM  "LT-7110 HI ALARM BIT" %
%   B3:0/1  ALARM_RESET  "ALARM RESET" %
%   B9:14/5  LT_7110_HI_ALT  "LT-7110 HI ALERT BIT" %
%   B3:0/0  ALARM_SILENCE  "ALARM SILENCE PUSHBUTTON" %
% Rung: 232 %
SOR GRT F8:28 F10:183 XIO B3:0/1 BST TON T4:183 1.0 0 0 NXB XIC T4:183/DN OSR B3:15/4 OTE B3:15/5 BND EOR
%   F8:28  LT_7110_SCI  "LT-7110 SCALED INPUT" %
%   F10:183  LT_7110_HIHI_SP  "LT-7110 HIHI ALARM SP" %
%   B3:0/1  ALARM_RESET  "ALARM RESET" %
%   T4:183  LT_7110_HIHI_DLY_TM  "LT-7110 HIHI ALARM DELAY" %
%   B3:15/4  "OSR" %
%   B3:15/5  "LT-7110 HIHI TRIGGER BIT" %
% Rung: 233 %
SOR BST BST XIC B3:15/5 NXB XIC B9:14/6 XIO B3:0/1 BND OTE B9:14/6 NXB BST XIC B3:15/5 NXB XIC B9:14/7 XIO B3:0/1 XIO B3:0/0 BND OTE B9:14/7 BND EOR
%   B3:15/5  "LT-7110 HIHI TRIGGER BIT" %
%   B9:14/6  LT_7110_HIHI_ALM  "LT-7110 HIHI ALARM BIT" %
%   B3:0/1  ALARM_RESET  "ALARM RESET" %
%   B9:14/7  LT_7110_HIHI_ALT  "LT-7110 HIHI ALERT BIT" %
%   B3:0/0  ALARM_SILENCE  "ALARM SILENCE PUSHBUTTON" %
% Rung: 234 %
SOR LES F8:29 F10:184 XIO B3:0/1 BST TON T4:184 1.0 10 10 NXB XIC T4:184/DN OSR B3:15/6 OTE B3:15/7 BND EOR
%   F8:29  LT_7130_SCI  "LT-7130 SCALED INPUT" %
%   F10:184  LT_7130_LOLO_SP  "LT-7130 LOLO ALARM SP" %
%   B3:0/1  ALARM_RESET  "ALARM RESET" %
%   T4:184  LT_7130_LOLO_DLY_TM  "LT-7130 LOLO ALARM DELAY" %
%   B3:15/6  "OSR" %
%   B3:15/7  "LT-7130 LOLO TRIGGER BIT" %

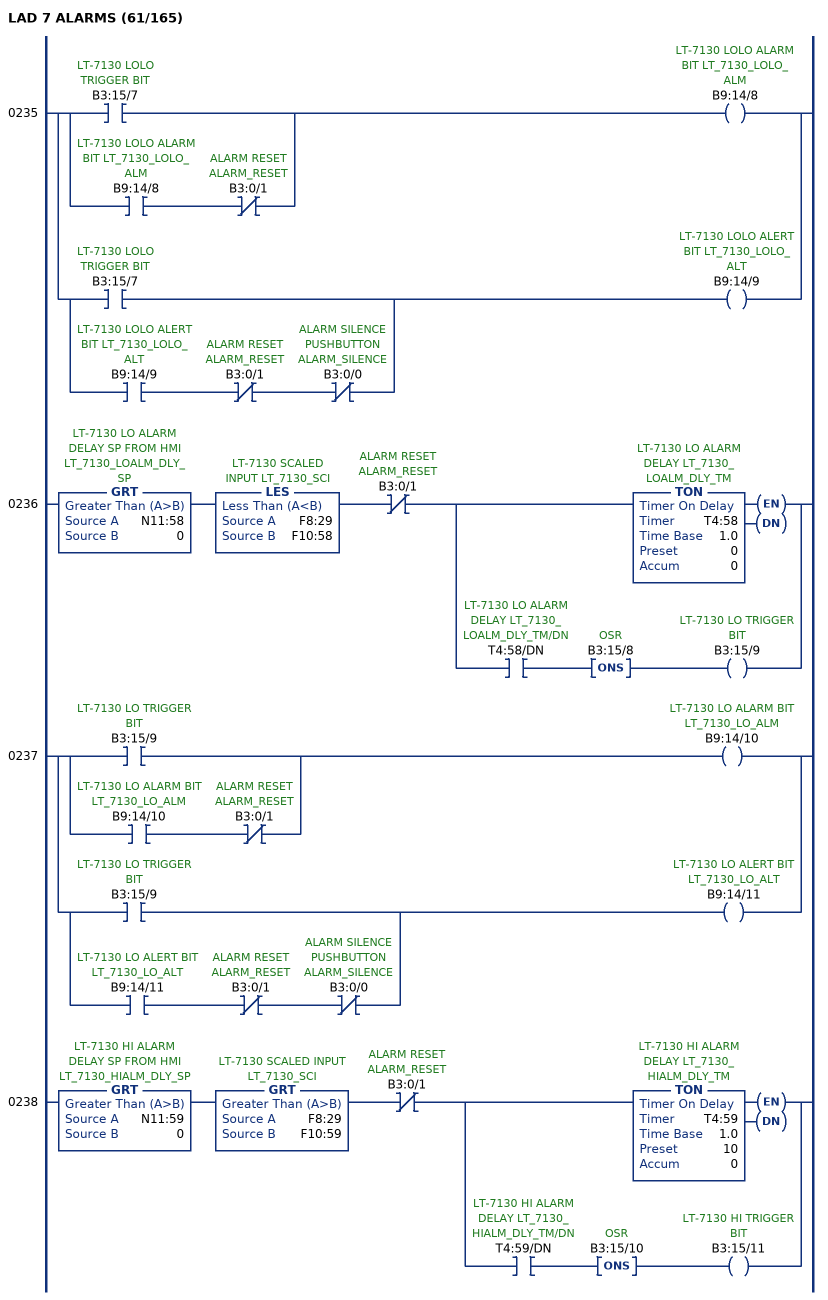
% Rung: 235 %
SOR BST BST XIC B3:15/7 NXB XIC B9:14/8 XIO B3:0/1 BND OTE B9:14/8 NXB BST XIC B3:15/7 NXB XIC B9:14/9 XIO B3:0/1 XIO B3:0/0 BND OTE B9:14/9 BND EOR
%   B3:15/7  "LT-7130 LOLO TRIGGER BIT" %
%   B9:14/8  LT_7130_LOLO_ALM  "LT-7130 LOLO ALARM BIT" %
%   B3:0/1  ALARM_RESET  "ALARM RESET" %
%   B9:14/9  LT_7130_LOLO_ALT  "LT-7130 LOLO ALERT BIT" %
%   B3:0/0  ALARM_SILENCE  "ALARM SILENCE PUSHBUTTON" %
% Rung: 236 %
SOR GRT N11:58 0 LES F8:29 F10:58 XIO B3:0/1 BST TON T4:58 1.0 0 0 NXB XIC T4:58/DN OSR B3:15/8 OTE B3:15/9 BND EOR
%   N11:58  LT_7130_LOALM_DLY_SP  "LT-7130 LO ALARM DELAY SP FROM HMI" %
%   F8:29  LT_7130_SCI  "LT-7130 SCALED INPUT" %
%   F10:58  LT_7130_LOALM_SP  "LT-7130 LO ALARM SP" %
%   B3:0/1  ALARM_RESET  "ALARM RESET" %
%   T4:58  LT_7130_LOALM_DLY_TM  "LT-7130 LO ALARM DELAY" %
%   B3:15/8  "OSR" %
%   B3:15/9  "LT-7130 LO TRIGGER BIT" %
% Rung: 237 %
SOR BST BST XIC B3:15/9 NXB XIC B9:14/10 XIO B3:0/1 BND OTE B9:14/10 NXB BST XIC B3:15/9 NXB XIC B9:14/11 XIO B3:0/1 XIO B3:0/0 BND OTE B9:14/11 BND EOR
%   B3:15/9  "LT-7130 LO TRIGGER BIT" %
%   B9:14/10  LT_7130_LO_ALM  "LT-7130 LO ALARM BIT" %
%   B3:0/1  ALARM_RESET  "ALARM RESET" %
%   B9:14/11  LT_7130_LO_ALT  "LT-7130 LO ALERT BIT" %
%   B3:0/0  ALARM_SILENCE  "ALARM SILENCE PUSHBUTTON" %
% Rung: 238 %
SOR GRT N11:59 0 GRT F8:29 F10:59 XIO B3:0/1 BST TON T4:59 1.0 10 0 NXB XIC T4:59/DN OSR B3:15/10 OTE B3:15/11 BND EOR
%   N11:59  LT_7130_HIALM_DLY_SP  "LT-7130 HI ALARM DELAY SP FROM HMI" %
%   F8:29  LT_7130_SCI  "LT-7130 SCALED INPUT" %
%   F10:59  LT_7130_HIALM_SP  "LT-7130 HI ALARM SP" %
%   B3:0/1  ALARM_RESET  "ALARM RESET" %
%   T4:59  LT_7130_HIALM_DLY_TM  "LT-7130 HI ALARM DELAY" %
%   B3:15/10  "OSR" %
%   B3:15/11  "LT-7130 HI TRIGGER BIT" %

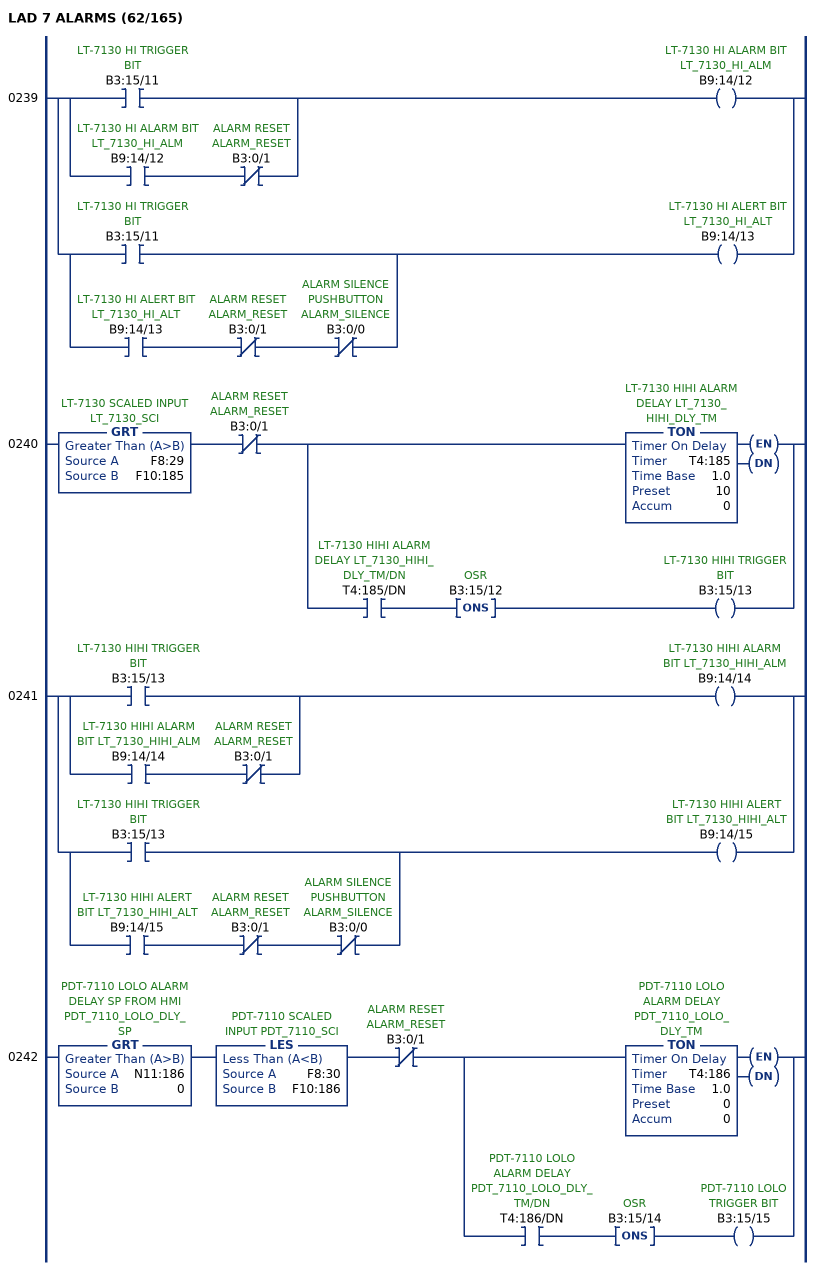
% Rung: 239 %
SOR BST BST XIC B3:15/11 NXB XIC B9:14/12 XIO B3:0/1 BND OTE B9:14/12 NXB BST XIC B3:15/11 NXB XIC B9:14/13 XIO B3:0/1 XIO B3:0/0 BND OTE B9:14/13 BND EOR
%   B3:15/11  "LT-7130 HI TRIGGER BIT" %
%   B9:14/12  LT_7130_HI_ALM  "LT-7130 HI ALARM BIT" %
%   B3:0/1  ALARM_RESET  "ALARM RESET" %
%   B9:14/13  LT_7130_HI_ALT  "LT-7130 HI ALERT BIT" %
%   B3:0/0  ALARM_SILENCE  "ALARM SILENCE PUSHBUTTON" %
% Rung: 240 %
SOR GRT F8:29 F10:185 XIO B3:0/1 BST TON T4:185 1.0 10 0 NXB XIC T4:185/DN OSR B3:15/12 OTE B3:15/13 BND EOR
%   F8:29  LT_7130_SCI  "LT-7130 SCALED INPUT" %
%   F10:185  LT_7130_HIHI_SP  "LT-7130 HIHI ALARM SP" %
%   B3:0/1  ALARM_RESET  "ALARM RESET" %
%   T4:185  LT_7130_HIHI_DLY_TM  "LT-7130 HIHI ALARM DELAY" %
%   B3:15/12  "OSR" %
%   B3:15/13  "LT-7130 HIHI TRIGGER BIT" %
% Rung: 241 %
SOR BST BST XIC B3:15/13 NXB XIC B9:14/14 XIO B3:0/1 BND OTE B9:14/14 NXB BST XIC B3:15/13 NXB XIC B9:14/15 XIO B3:0/1 XIO B3:0/0 BND OTE B9:14/15 BND EOR
%   B3:15/13  "LT-7130 HIHI TRIGGER BIT" %
%   B9:14/14  LT_7130_HIHI_ALM  "LT-7130 HIHI ALARM BIT" %
%   B3:0/1  ALARM_RESET  "ALARM RESET" %
%   B9:14/15  LT_7130_HIHI_ALT  "LT-7130 HIHI ALERT BIT" %
%   B3:0/0  ALARM_SILENCE  "ALARM SILENCE PUSHBUTTON" %
% Rung: 242 %
SOR GRT N11:186 0 LES F8:30 F10:186 XIO B3:0/1 BST TON T4:186 1.0 0 0 NXB XIC T4:186/DN OSR B3:15/14 OTE B3:15/15 BND EOR
%   N11:186  PDT_7110_LOLO_DLY_SP  "PDT-7110 LOLO ALARM DELAY SP FROM HMI" %
%   F8:30  PDT_7110_SCI  "PDT-7110 SCALED INPUT" %
%   F10:186  PDT_7110_LOLO_SP  "PDT-7110 LOLO ALARM SP" %
%   B3:0/1  ALARM_RESET  "ALARM RESET" %
%   T4:186  PDT_7110_LOLO_DLY_TM  "PDT-7110 LOLO ALARM DELAY" %
%   B3:15/14  "OSR" %
%   B3:15/15  "PDT-7110 LOLO TRIGGER BIT" %

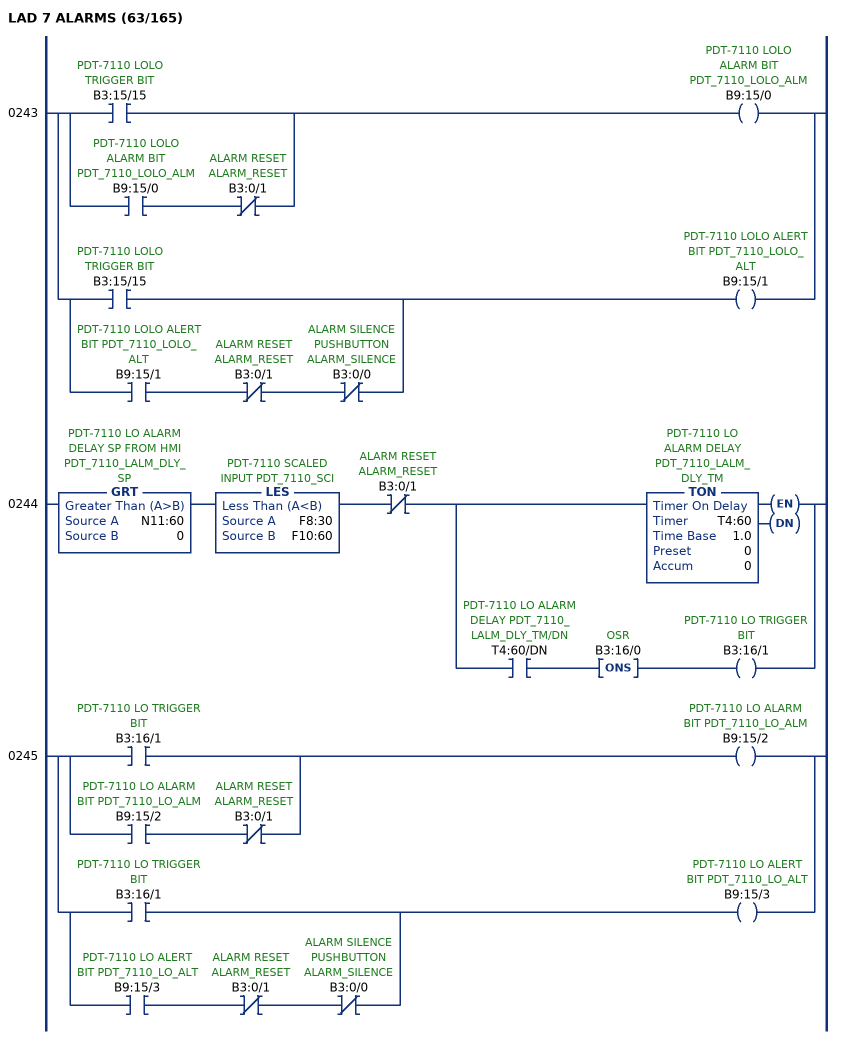
% Rung: 243 %
SOR BST BST XIC B3:15/15 NXB XIC B9:15/0 XIO B3:0/1 BND OTE B9:15/0 NXB BST XIC B3:15/15 NXB XIC B9:15/1 XIO B3:0/1 XIO B3:0/0 BND OTE B9:15/1 BND EOR
%   B3:15/15  "PDT-7110 LOLO TRIGGER BIT" %
%   B9:15/0  PDT_7110_LOLO_ALM  "PDT-7110 LOLO ALARM BIT" %
%   B3:0/1  ALARM_RESET  "ALARM RESET" %
%   B9:15/1  PDT_7110_LOLO_ALT  "PDT-7110 LOLO ALERT BIT" %
%   B3:0/0  ALARM_SILENCE  "ALARM SILENCE PUSHBUTTON" %
% Rung: 244 %
SOR GRT N11:60 0 LES F8:30 F10:60 XIO B3:0/1 BST TON T4:60 1.0 0 0 NXB XIC T4:60/DN OSR B3:16/0 OTE B3:16/1 BND EOR
%   N11:60  PDT_7110_LALM_DLY_SP  "PDT-7110 LO ALARM DELAY SP FROM HMI" %
%   F8:30  PDT_7110_SCI  "PDT-7110 SCALED INPUT" %
%   F10:60  PDT_7110_LOALM_SP  "PDT-7110 LO ALARM SP" %
%   B3:0/1  ALARM_RESET  "ALARM RESET" %
%   T4:60  PDT_7110_LALM_DLY_TM  "PDT-7110 LO ALARM DELAY" %
%   B3:16/0  "OSR" %
%   B3:16/1  "PDT-7110 LO TRIGGER BIT" %
% Rung: 245 %
SOR BST BST XIC B3:16/1 NXB XIC B9:15/2 XIO B3:0/1 BND OTE B9:15/2 NXB BST XIC B3:16/1 NXB XIC B9:15/3 XIO B3:0/1 XIO B3:0/0 BND OTE B9:15/3 BND EOR
%   B3:16/1  "PDT-7110 LO TRIGGER BIT" %
%   B9:15/2  PDT_7110_LO_ALM  "PDT-7110 LO ALARM BIT" %
%   B3:0/1  ALARM_RESET  "ALARM RESET" %
%   B9:15/3  PDT_7110_LO_ALT  "PDT-7110 LO ALERT BIT" %
%   B3:0/0  ALARM_SILENCE  "ALARM SILENCE PUSHBUTTON" %

